// TIA Portal V16 export
// export: Created 2021-11-12T13:31:13.1674631Z, ExportSetting WithDefaults, DisplayName Totally Integrated Automation Portal, DisplayVersion V16 Update 3, DisplayName TIA Portal Version Control Interface, DisplayVersion V16 Update 2, DisplayName TIA Portal Openness, DisplayVersion V16 Update 3, DisplayName SINAMICS Startdrive Advanced, DisplayVersion V16 Update 5, DisplayName SINAMICS Startdrive G130, G150, S120, S150, SINAMICS MV, S210, DisplayVersion V16 Update 5, DisplayName SINAMICS Startdrive G110M, G120, G120C, G120D, G120P, G115D, DisplayVersion V16 Update 5, DisplayName STEP 7 Professional, DisplayVersion V16 Update 3, DisplayName STEP 7 Safety, DisplayVersion V16, DisplayName WinCC UA Professional, DisplayVersion V16 Update 3
FUNCTION_BLOCK "STD_RobotGripper"   // FB1227, LAD
{ S7_Optimized_Access := 'TRUE' }
VERSION : 0.1
// MICE STD Function block
// STD_RobotGripper
// 
// Version      Creation date        Created by
// 1.0                 24.9.2018                   RS
// stored: AutoNumber false, IsIECCheckEnabled false, IsRetainMemResEnabled false, MemoryReserve 100, SetENOAutomatically false, UDAEnableTagReadback false
   VAR_INPUT
      IS_Gripper : "UDT_RobotGripper_Inputs";
      IS_ZoneM { ExternalAccessible := 'False'; ExternalVisible := 'False'; ExternalWritable := 'False'} : "UDT_Status_main";   // Main structure from zone
      IS_ZoneS { ExternalAccessible := 'False'; ExternalVisible := 'False'; ExternalWritable := 'False'} : "UDT_Zone_Status_specific";   // Specific structure from zone
      IB1AlarmSuppress : Bool;   // Suppress alarms
      IT_AckPulseTime : Time := T#200ms;   // Acknowledge pulse length
   END_VAR
   VAR_OUTPUT
      OS_Status : Struct
         Main : "UDT_Status_main";
         Specific : "UDT_RobotGripper_Status_specific";
         Error : "UDT_Error10";
      END_STRUCT;
      OS_Gripper : "UDT_RobotGripper_Outputs";
   END_VAR
   VAR_IN_OUT
      XS_Command : "UDT_RobotGripper_Command";
      XS_Parameter : "UDT_RobotGripper_Parameter";
   END_VAR
   VAR
      SS_Alarm : Struct   // Device alarms / Alarmy zařízení
         MediaNotOK : Bool;   // Gripper media is not OK / Chyba gripperu - nesoulad mezi skutečným a očekávaným stavem
         Res_00_1 : Bool;   // Chyba kontroléru robota - více informací lze nalézt na teachpendantu robota
         Res_00_2 : Bool;   // Chyba robota - více informací lze nalézt na teachpendantu robota
         Res_00_3 : Bool;   // Stisknuto tlačítko Estop na robotu
         Res_00_4 : Bool;   // Bezpečnostní okruh robota přerušen
         Res_00_5 : Bool;   // Motion supervision detekovat kolizi robota
         Res_00_6 : Bool;   // Zpětná vazba čísla úlohy robota neodpovídá požadavku
         Res_00_7 : Bool;   // Zpětná vazba čísla typu úlohy robota neodpovídá požadavku
         Res_01_0 : Bool;
         Res_01_1 : Bool;
         Res_01_2 : Bool;
         Res_01_3 : Bool;
         Res_01_4 : Bool;
         Res_01_5 : Bool;
         Res_01_6 : Bool;
         Res_01_7 : Bool;
      END_STRUCT;
      SS_Warning : Struct   // Device warnings / Varovaní zařízení
         GripperError : Bool;   // Gripper - discrepancy between real and expected state / Chyba gripperu - nesoulad mezi skutečným a očekávaným stavem
         IgnoreGripperError : Bool;   // Gripper error not evaluated / Rychlost robota je omezena na bezpečnou (250mm/s)
         Res_00_2 : Bool;   // Varování robota - více informací lze nalézt na teachpendantu robota
         Res_00_3 : Bool;   // Dialogové okno na Teachpendantu vyžaduje interakci uživatele
         Res_00_4 : Bool;
         Res_00_5 : Bool;
         Res_00_6 : Bool;
         Res_00_7 : Bool;
         Res_01_0 : Bool;
         Res_01_1 : Bool;
         Res_01_2 : Bool;
         Res_01_3 : Bool;
         Res_01_4 : Bool;
         Res_01_5 : Bool;
         Res_01_6 : Bool;
         Res_01_7 : Bool;
         Positive_00_00 : Bool;   // Gripper signal 0 missing
         Positive_00_01 : Bool;   // Gripper signal 1 missing
         Positive_00_02 : Bool;   // Gripper signal 2 missing
         Positive_00_03 : Bool;   // Gripper signal 3 missing
         Positive_00_04 : Bool;   // Gripper signal 4 missing
         Positive_00_05 : Bool;   // Gripper signal 5 missing
         Positive_00_06 : Bool;   // Gripper signal 6 missing
         Positive_00_07 : Bool;   // Gripper signal 7 missing
         Positive_00_08 : Bool;   // Gripper signal 8 missing
         Positive_00_09 : Bool;   // Gripper signal 9 missing
         Positive_00_10 : Bool;   // Gripper signal 10 missing
         Positive_00_11 : Bool;   // Gripper signal 11 missing
         Positive_00_12 : Bool;   // Gripper signal 12 missing
         Positive_00_13 : Bool;   // Gripper signal 13 missing
         Positive_00_14 : Bool;   // Gripper signal 14 missing
         Positive_00_15 : Bool;   // Gripper signal 15 missing
         Positive_00_16 : Bool;   // Gripper signal 16 missing
         Positive_00_17 : Bool;   // Gripper signal 17 missing
         Positive_00_18 : Bool;   // Gripper signal 18 missing
         Positive_00_19 : Bool;   // Gripper signal 19 missing
         Positive_00_20 : Bool;   // Gripper signal 20 missing
         Positive_00_21 : Bool;   // Gripper signal 21 missing
         Positive_00_22 : Bool;   // Gripper signal 22 missing
         Positive_00_23 : Bool;   // Gripper signal 23 missing
         Positive_00_24 : Bool;   // Gripper signal 24 missing
         Positive_00_25 : Bool;   // Gripper signal 25 missing
         Positive_00_26 : Bool;   // Gripper signal 26 missing
         Positive_00_27 : Bool;   // Gripper signal 27 missing
         Positive_00_28 : Bool;   // Gripper signal 28 missing
         Positive_00_29 : Bool;   // Gripper signal 29 missing
         Positive_00_30 : Bool;   // Gripper signal 30 missing
         Positive_00_31 : Bool;   // Gripper signal 31 missing
         Negative_00_00 : Bool;   // Gripper signal 0 is true
         Negative_00_01 : Bool;   // Gripper signal 1 is true
         Negative_00_02 : Bool;   // Gripper signal 2 is true
         Negative_00_03 : Bool;   // Gripper signal 3 is true
         Negative_00_04 : Bool;   // Gripper signal 4 is true
         Negative_00_05 : Bool;   // Gripper signal 5 is true
         Negative_00_06 : Bool;   // Gripper signal 6 is true
         Negative_00_07 : Bool;   // Gripper signal 7 is true
         Negative_00_08 : Bool;   // Gripper signal 8 is true
         Negative_00_09 : Bool;   // Gripper signal 9 is true
         Negative_00_10 : Bool;   // Gripper signal 10 is true
         Negative_00_11 : Bool;   // Gripper signal 11 is true
         Negative_00_12 : Bool;   // Gripper signal 12 is true
         Negative_00_13 : Bool;   // Gripper signal 13 is true
         Negative_00_14 : Bool;   // Gripper signal 14 is true
         Negative_00_15 : Bool;   // Gripper signal 15 is true
         Negative_00_16 : Bool;   // Gripper signal 16 is true
         Negative_00_17 : Bool;   // Gripper signal 17 is true
         Negative_00_18 : Bool;   // Gripper signal 18 is true
         Negative_00_19 : Bool;   // Gripper signal 19 is true
         Negative_00_20 : Bool;   // Gripper signal 20 is true
         Negative_00_21 : Bool;   // Gripper signal 21 is true
         Negative_00_22 : Bool;   // Gripper signal 22 is true
         Negative_00_23 : Bool;   // Gripper signal 23 is true
         Negative_00_24 : Bool;   // Gripper signal 24 is true
         Negative_00_25 : Bool;   // Gripper signal 25 is true
         Negative_00_26 : Bool;   // Gripper signal 26 is true
         Negative_00_27 : Bool;   // Gripper signal 27 is true
         Negative_00_28 : Bool;   // Gripper signal 28 is true
         Negative_00_29 : Bool;   // Gripper signal 29 is true
         Negative_00_30 : Bool;   // Gripper signal 30 is true
         Negative_00_31 : Bool;   // Gripper signal 31 is true
      END_STRUCT;
      SS_Input : Struct
         Gripper { S7_SetPoint := 'True'} : "UDT_RobotGripper_Inputs";
      END_STRUCT;
      SS_Output : Struct
         Gripper { S7_SetPoint := 'True'} : "UDT_RobotGripper_Outputs";
      END_STRUCT;
      SB1IgnoreGripperError : Bool;
      ST_ResetError_TOF { S7_SetPoint := 'True'} : TOF_TIME;
      ST_ResetError_TP { S7_SetPoint := 'True'} : TP_TIME;
      ST_Retest_TOF { S7_SetPoint := 'True'} : TOF_TIME;
      ST_Retry_TOF { S7_SetPoint := 'True'} : TOF_TIME;
   END_VAR
   VAR_TEMP
      TS_Status : Struct
         Main : "UDT_Status_main";
         Specific : "UDT_RobotGripper_Status_specific";
         Error : "UDT_Error10";
      END_STRUCT;
      TS_Parameter : "UDT_RobotGripper_Parameter";
      TS_Command : "UDT_RobotGripper_Command";
      TB1AckPulse : Bool;
      TD_XOR : DWord;
   END_VAR
   VAR_TEMP   // added for the SCL form of the ladder/FBD networks
      _w1 : Bool;
      _w2 : Bool;
      _w3 : Bool;
      _w4 : Bool;
      _w5 : Bool;
      _w6 : Bool;
      _w7 : Bool;
      _w8 : Bool;
      _w9 : Bool;
      _w10 : Bool;
      _w11 : Bool;
      _w12 : Bool;
      _w13 : Bool;
      _w14 : Bool;
      _w15 : Bool;
      _w16 : Bool;
      _w17 : Bool;
      _w18 : Bool;
      _w19 : Bool;
      _w20 : Bool;
      _w21 : Bool;
      _w22 : Bool;
      _w23 : Bool;
      _w24 : Bool;
      _w25 : Bool;
      _w26 : Bool;
      _w27 : Bool;
      _w28 : Bool;
      _w29 : Bool;
      _w30 : Bool;
      _w31 : Bool;
      _w32 : Bool;
   END_VAR
BEGIN

REGION Network 1: Clear temporary TS_Status - Main, Specific
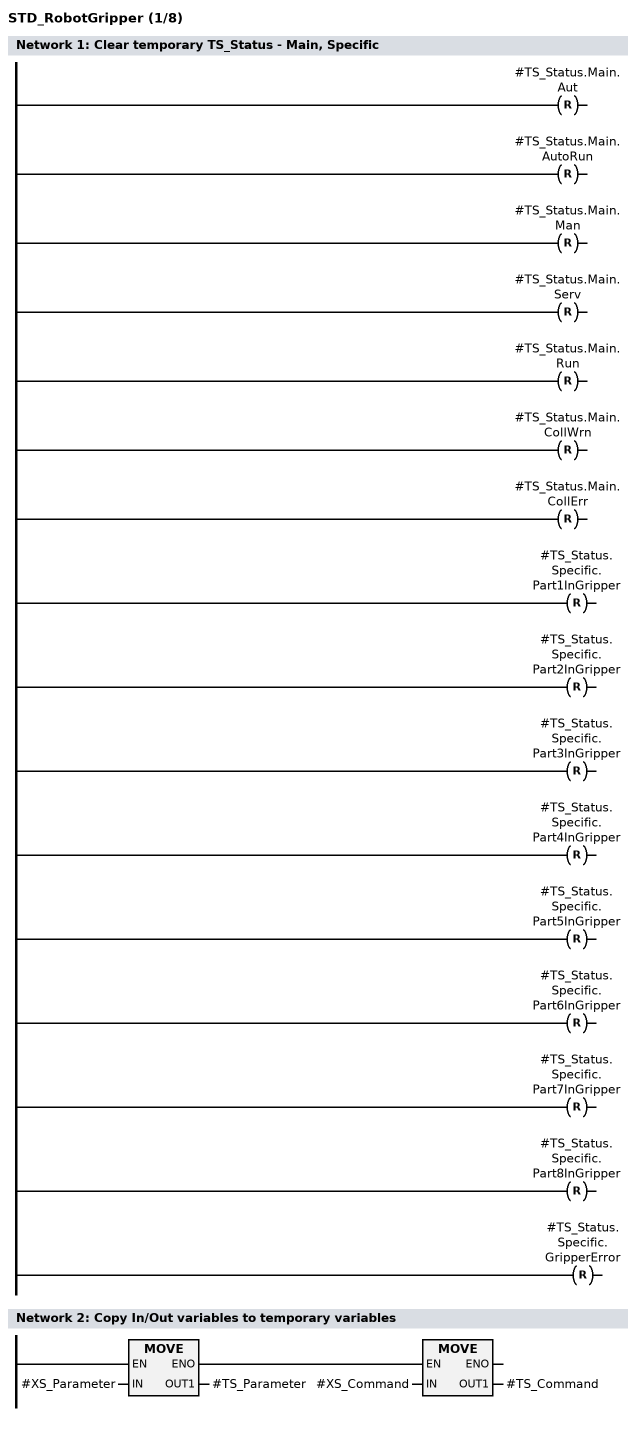
   RUNG wire#powerrail
      R_Coil( #TS_Status.Main.Aut )
   END_RUNG
   RUNG wire#powerrail
      R_Coil( #TS_Status.Main.AutoRun )
   END_RUNG
   RUNG wire#powerrail
      R_Coil( #TS_Status.Main.Man )
   END_RUNG
   RUNG wire#powerrail
      R_Coil( #TS_Status.Main.Serv )
   END_RUNG
   RUNG wire#powerrail
      R_Coil( #TS_Status.Main.Run )
   END_RUNG
   RUNG wire#powerrail
      R_Coil( #TS_Status.Main.CollWrn )
   END_RUNG
   RUNG wire#powerrail
      R_Coil( #TS_Status.Main.CollErr )
   END_RUNG
   RUNG wire#powerrail
      R_Coil( #TS_Status.Specific.Part1InGripper )
   END_RUNG
   RUNG wire#powerrail
      R_Coil( #TS_Status.Specific.Part2InGripper )
   END_RUNG
   RUNG wire#powerrail
      R_Coil( #TS_Status.Specific.Part3InGripper )
   END_RUNG
   RUNG wire#powerrail
      R_Coil( #TS_Status.Specific.Part4InGripper )
   END_RUNG
   RUNG wire#powerrail
      R_Coil( #TS_Status.Specific.Part5InGripper )
   END_RUNG
   RUNG wire#powerrail
      R_Coil( #TS_Status.Specific.Part6InGripper )
   END_RUNG
   RUNG wire#powerrail
      R_Coil( #TS_Status.Specific.Part7InGripper )
   END_RUNG
   RUNG wire#powerrail
      R_Coil( #TS_Status.Specific.Part8InGripper )
   END_RUNG
   RUNG wire#powerrail
      R_Coil( #TS_Status.Specific.GripperError )
   END_RUNG
   // the same network as SCL:
   #TS_Status.Main.Aut := FALSE;
   #TS_Status.Main.AutoRun := FALSE;
   #TS_Status.Main.Man := FALSE;
   #TS_Status.Main.Serv := FALSE;
   #TS_Status.Main.Run := FALSE;
   #TS_Status.Main.CollWrn := FALSE;
   #TS_Status.Main.CollErr := FALSE;
   #TS_Status.Specific.Part1InGripper := FALSE;
   #TS_Status.Specific.Part2InGripper := FALSE;
   #TS_Status.Specific.Part3InGripper := FALSE;
   #TS_Status.Specific.Part4InGripper := FALSE;
   #TS_Status.Specific.Part5InGripper := FALSE;
   #TS_Status.Specific.Part6InGripper := FALSE;
   #TS_Status.Specific.Part7InGripper := FALSE;
   #TS_Status.Specific.Part8InGripper := FALSE;
   #TS_Status.Specific.GripperError := FALSE;
END_REGION

REGION Network 2: Copy In/Out variables to temporary variables
   RUNG wire#powerrail
      Move(in := #XS_Parameter, out1 => #TS_Parameter)
      Move(in := #XS_Command, out1 => #TS_Command)
   END_RUNG
   // the same network as SCL:
   #TS_Parameter := #XS_Parameter;
   #TS_Command := #XS_Command;
END_REGION

REGION Network 3: Read data from Robot Interface
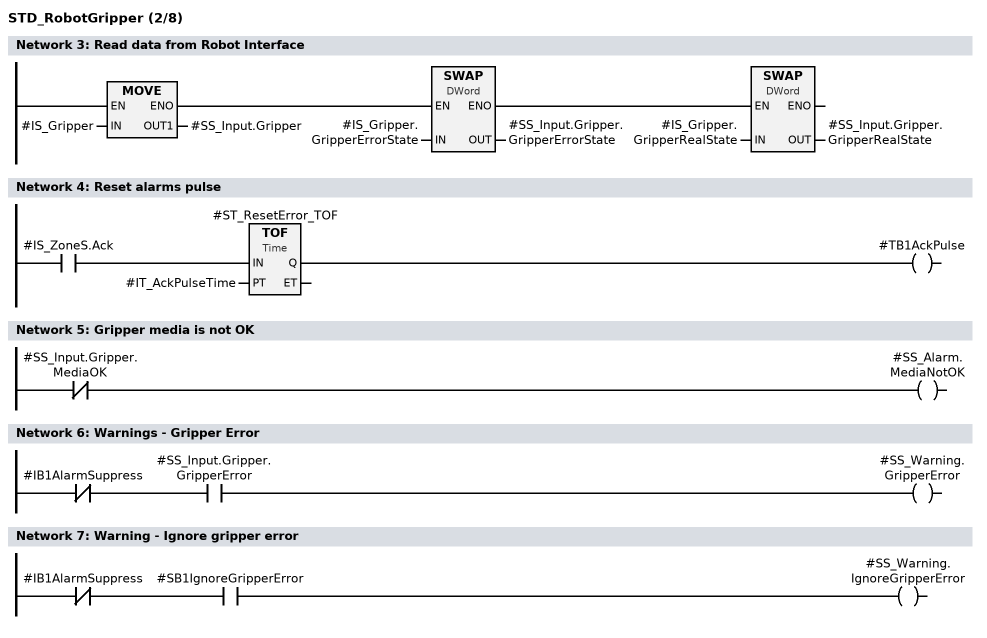
   #SS_Input.Gripper := #IS_Gripper;
   #SS_Input.Gripper.GripperErrorState := SWAP(#IS_Gripper.GripperErrorState);
   #SS_Input.Gripper.GripperRealState := SWAP(#IS_Gripper.GripperRealState);
END_REGION

REGION Network 4: Reset alarms pulse
   RUNG wire#powerrail
      Contact( #IS_ZoneS.Ack )
      { S7_Templates := "time_type := Time" } #ST_ResetError_TOF.TOF(pt := #IT_AckPulseTime, et =>)
      Coil( #TB1AckPulse )
   END_RUNG
   // the same network as SCL:
   #ST_ResetError_TOF(IN := #IS_ZoneS.Ack, PT := #IT_AckPulseTime);   // TOF
   #TB1AckPulse := #ST_ResetError_TOF.Q;
END_REGION

REGION Network 5: Gripper media is not OK
   RUNG wire#powerrail
      I_Contact( #SS_Input.Gripper.MediaOK )
      Coil( #SS_Alarm.MediaNotOK )
   END_RUNG
   // the same network as SCL:
   #SS_Alarm.MediaNotOK := NOT #SS_Input.Gripper.MediaOK;
END_REGION

REGION Network 6: Warnings - Gripper Error
   RUNG wire#powerrail
      I_Contact( #IB1AlarmSuppress )
      Contact( #SS_Input.Gripper.GripperError )
      Coil( #SS_Warning.GripperError )
   END_RUNG
   // the same network as SCL:
   #SS_Warning.GripperError := NOT #IB1AlarmSuppress AND #SS_Input.Gripper.GripperError;
END_REGION

REGION Network 7: Warning - Ignore gripper error
   RUNG wire#powerrail
      I_Contact( #IB1AlarmSuppress )
      Contact( #SB1IgnoreGripperError )
      Coil( #SS_Warning.IgnoreGripperError )
   END_RUNG
   // the same network as SCL:
   #SS_Warning.IgnoreGripperError := NOT #IB1AlarmSuppress AND #SB1IgnoreGripperError;
END_REGION

REGION Network 8: Gripper Specific error
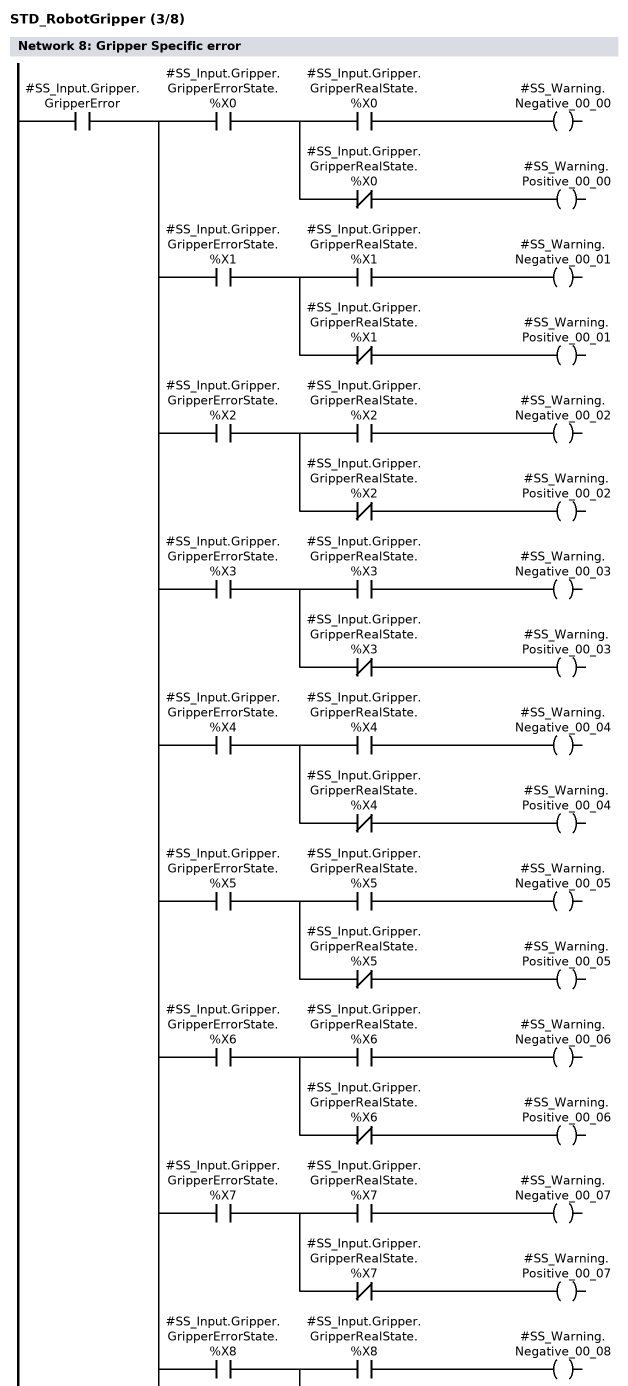
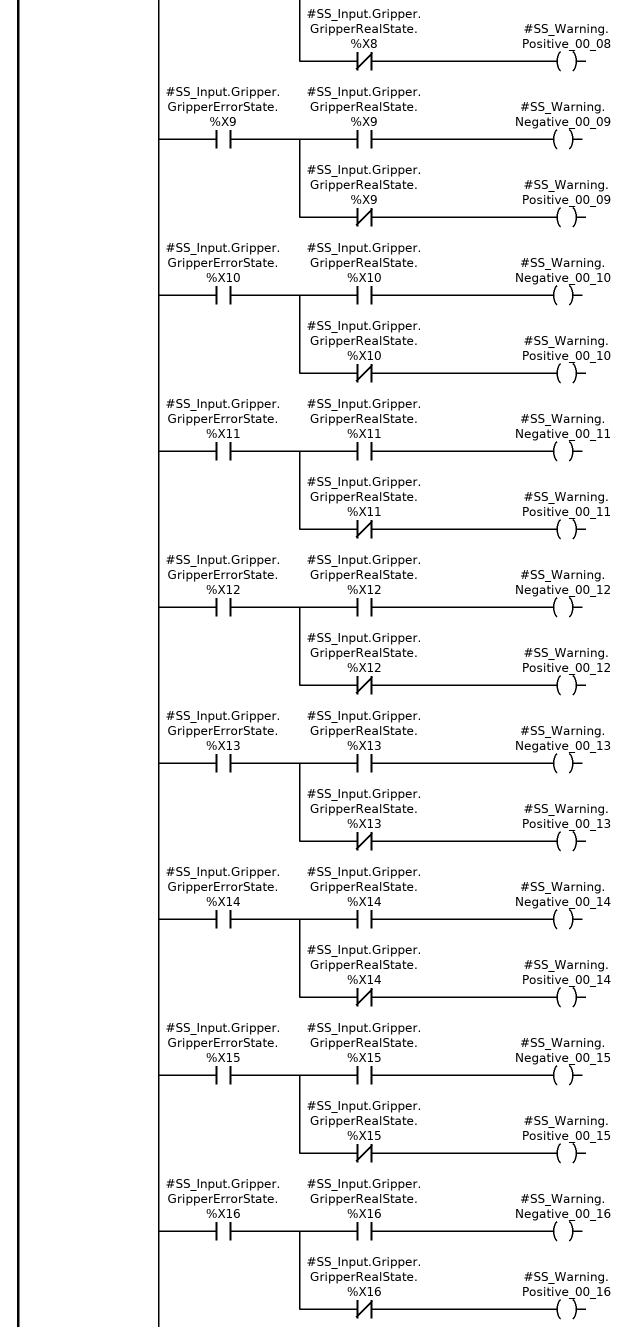
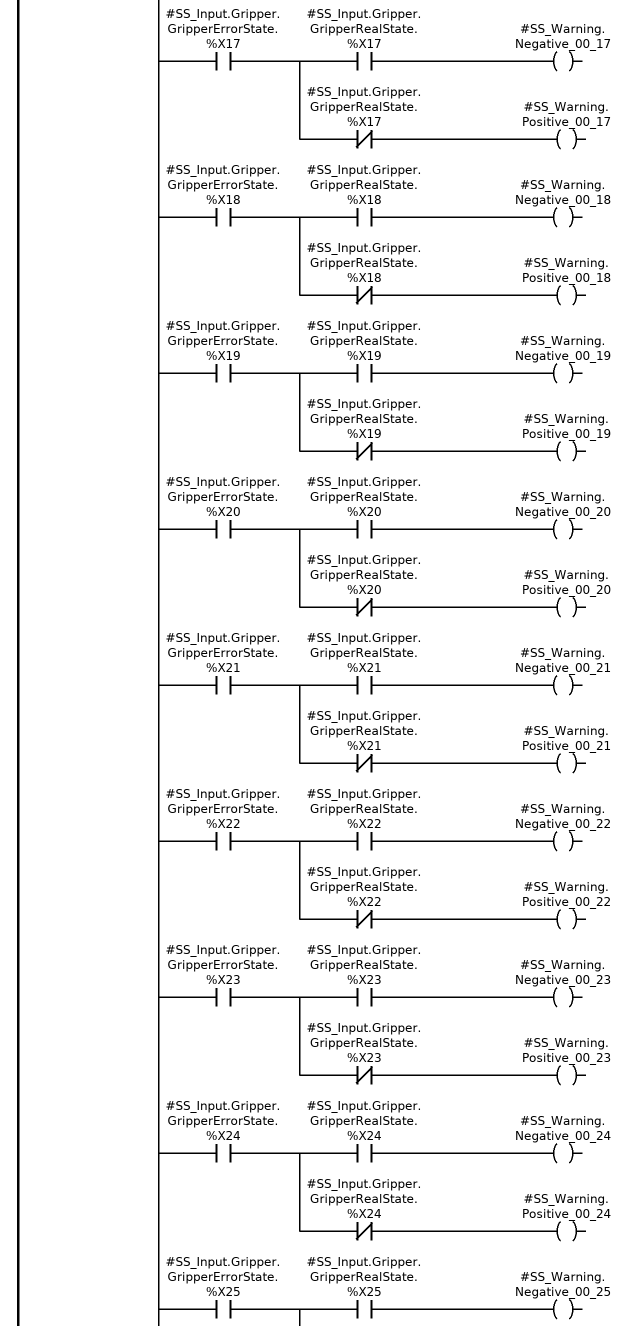
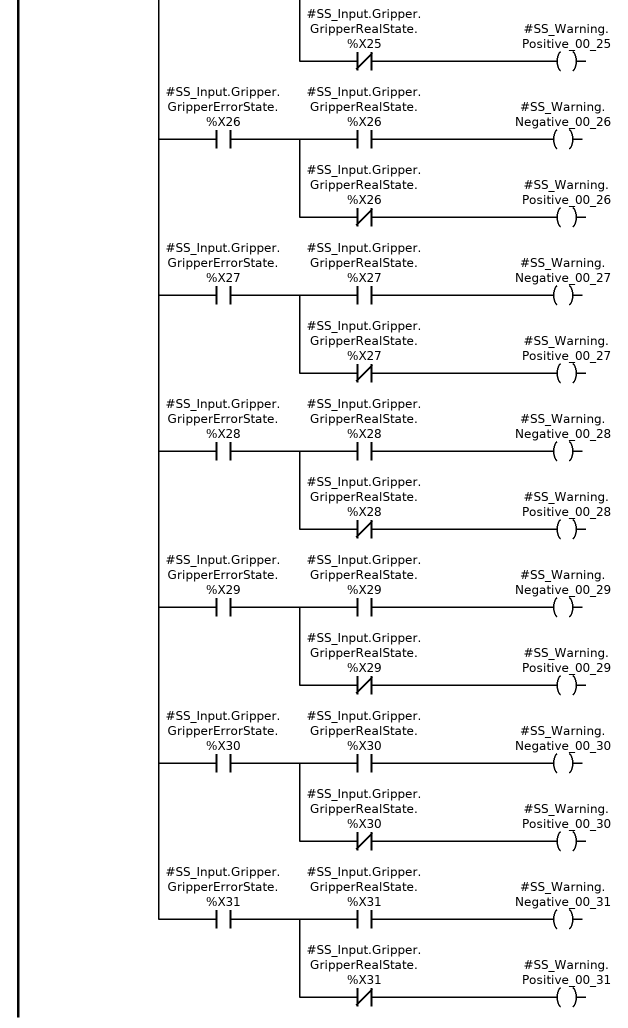
   RUNG wire#powerrail
      Contact( #SS_Input.Gripper.GripperError )
      wire#w1
      Contact( #SS_Input.Gripper.GripperErrorState.%X0 )
      wire#w2
      Contact( #SS_Input.Gripper.GripperRealState.%X0 )
      Coil( #SS_Warning.Negative_00_00 )
   END_RUNG
   RUNG wire#w2
      I_Contact( #SS_Input.Gripper.GripperRealState.%X0 )
      Coil( #SS_Warning.Positive_00_00 )
   END_RUNG
   RUNG wire#w1
      Contact( #SS_Input.Gripper.GripperErrorState.%X1 )
      wire#w3
      Contact( #SS_Input.Gripper.GripperRealState.%X1 )
      Coil( #SS_Warning.Negative_00_01 )
   END_RUNG
   RUNG wire#w3
      I_Contact( #SS_Input.Gripper.GripperRealState.%X1 )
      Coil( #SS_Warning.Positive_00_01 )
   END_RUNG
   RUNG wire#w1
      Contact( #SS_Input.Gripper.GripperErrorState.%X2 )
      wire#w4
      Contact( #SS_Input.Gripper.GripperRealState.%X2 )
      Coil( #SS_Warning.Negative_00_02 )
   END_RUNG
   RUNG wire#w4
      I_Contact( #SS_Input.Gripper.GripperRealState.%X2 )
      Coil( #SS_Warning.Positive_00_02 )
   END_RUNG
   RUNG wire#w1
      Contact( #SS_Input.Gripper.GripperErrorState.%X3 )
      wire#w5
      Contact( #SS_Input.Gripper.GripperRealState.%X3 )
      Coil( #SS_Warning.Negative_00_03 )
   END_RUNG
   RUNG wire#w5
      I_Contact( #SS_Input.Gripper.GripperRealState.%X3 )
      Coil( #SS_Warning.Positive_00_03 )
   END_RUNG
   RUNG wire#w1
      Contact( #SS_Input.Gripper.GripperErrorState.%X4 )
      wire#w6
      Contact( #SS_Input.Gripper.GripperRealState.%X4 )
      Coil( #SS_Warning.Negative_00_04 )
   END_RUNG
   RUNG wire#w6
      I_Contact( #SS_Input.Gripper.GripperRealState.%X4 )
      Coil( #SS_Warning.Positive_00_04 )
   END_RUNG
   RUNG wire#w1
      Contact( #SS_Input.Gripper.GripperErrorState.%X5 )
      wire#w7
      Contact( #SS_Input.Gripper.GripperRealState.%X5 )
      Coil( #SS_Warning.Negative_00_05 )
   END_RUNG
   RUNG wire#w7
      I_Contact( #SS_Input.Gripper.GripperRealState.%X5 )
      Coil( #SS_Warning.Positive_00_05 )
   END_RUNG
   RUNG wire#w1
      Contact( #SS_Input.Gripper.GripperErrorState.%X6 )
      wire#w8
      Contact( #SS_Input.Gripper.GripperRealState.%X6 )
      Coil( #SS_Warning.Negative_00_06 )
   END_RUNG
   RUNG wire#w8
      I_Contact( #SS_Input.Gripper.GripperRealState.%X6 )
      Coil( #SS_Warning.Positive_00_06 )
   END_RUNG
   RUNG wire#w1
      Contact( #SS_Input.Gripper.GripperErrorState.%X7 )
      wire#w9
      Contact( #SS_Input.Gripper.GripperRealState.%X7 )
      Coil( #SS_Warning.Negative_00_07 )
   END_RUNG
   RUNG wire#w9
      I_Contact( #SS_Input.Gripper.GripperRealState.%X7 )
      Coil( #SS_Warning.Positive_00_07 )
   END_RUNG
   RUNG wire#w1
      Contact( #SS_Input.Gripper.GripperErrorState.%X8 )
      wire#w10
      Contact( #SS_Input.Gripper.GripperRealState.%X8 )
      Coil( #SS_Warning.Negative_00_08 )
   END_RUNG
   RUNG wire#w10
      I_Contact( #SS_Input.Gripper.GripperRealState.%X8 )
      Coil( #SS_Warning.Positive_00_08 )
   END_RUNG
   RUNG wire#w1
      Contact( #SS_Input.Gripper.GripperErrorState.%X9 )
      wire#w11
      Contact( #SS_Input.Gripper.GripperRealState.%X9 )
      Coil( #SS_Warning.Negative_00_09 )
   END_RUNG
   RUNG wire#w11
      I_Contact( #SS_Input.Gripper.GripperRealState.%X9 )
      Coil( #SS_Warning.Positive_00_09 )
   END_RUNG
   RUNG wire#w1
      Contact( #SS_Input.Gripper.GripperErrorState.%X10 )
      wire#w12
      Contact( #SS_Input.Gripper.GripperRealState.%X10 )
      Coil( #SS_Warning.Negative_00_10 )
   END_RUNG
   RUNG wire#w12
      I_Contact( #SS_Input.Gripper.GripperRealState.%X10 )
      Coil( #SS_Warning.Positive_00_10 )
   END_RUNG
   RUNG wire#w1
      Contact( #SS_Input.Gripper.GripperErrorState.%X11 )
      wire#w13
      Contact( #SS_Input.Gripper.GripperRealState.%X11 )
      Coil( #SS_Warning.Negative_00_11 )
   END_RUNG
   RUNG wire#w13
      I_Contact( #SS_Input.Gripper.GripperRealState.%X11 )
      Coil( #SS_Warning.Positive_00_11 )
   END_RUNG
   RUNG wire#w1
      Contact( #SS_Input.Gripper.GripperErrorState.%X12 )
      wire#w14
      Contact( #SS_Input.Gripper.GripperRealState.%X12 )
      Coil( #SS_Warning.Negative_00_12 )
   END_RUNG
   RUNG wire#w14
      I_Contact( #SS_Input.Gripper.GripperRealState.%X12 )
      Coil( #SS_Warning.Positive_00_12 )
   END_RUNG
   RUNG wire#w1
      Contact( #SS_Input.Gripper.GripperErrorState.%X13 )
      wire#w15
      Contact( #SS_Input.Gripper.GripperRealState.%X13 )
      Coil( #SS_Warning.Negative_00_13 )
   END_RUNG
   RUNG wire#w15
      I_Contact( #SS_Input.Gripper.GripperRealState.%X13 )
      Coil( #SS_Warning.Positive_00_13 )
   END_RUNG
   RUNG wire#w1
      Contact( #SS_Input.Gripper.GripperErrorState.%X14 )
      wire#w16
      Contact( #SS_Input.Gripper.GripperRealState.%X14 )
      Coil( #SS_Warning.Negative_00_14 )
   END_RUNG
   RUNG wire#w16
      I_Contact( #SS_Input.Gripper.GripperRealState.%X14 )
      Coil( #SS_Warning.Positive_00_14 )
   END_RUNG
   RUNG wire#w1
      Contact( #SS_Input.Gripper.GripperErrorState.%X15 )
      wire#w17
      Contact( #SS_Input.Gripper.GripperRealState.%X15 )
      Coil( #SS_Warning.Negative_00_15 )
   END_RUNG
   RUNG wire#w17
      I_Contact( #SS_Input.Gripper.GripperRealState.%X15 )
      Coil( #SS_Warning.Positive_00_15 )
   END_RUNG
   RUNG wire#w1
      Contact( #SS_Input.Gripper.GripperErrorState.%X16 )
      wire#w18
      Contact( #SS_Input.Gripper.GripperRealState.%X16 )
      Coil( #SS_Warning.Negative_00_16 )
   END_RUNG
   RUNG wire#w18
      I_Contact( #SS_Input.Gripper.GripperRealState.%X16 )
      Coil( #SS_Warning.Positive_00_16 )
   END_RUNG
   RUNG wire#w1
      Contact( #SS_Input.Gripper.GripperErrorState.%X17 )
      wire#w19
      Contact( #SS_Input.Gripper.GripperRealState.%X17 )
      Coil( #SS_Warning.Negative_00_17 )
   END_RUNG
   RUNG wire#w19
      I_Contact( #SS_Input.Gripper.GripperRealState.%X17 )
      Coil( #SS_Warning.Positive_00_17 )
   END_RUNG
   RUNG wire#w1
      Contact( #SS_Input.Gripper.GripperErrorState.%X18 )
      wire#w20
      Contact( #SS_Input.Gripper.GripperRealState.%X18 )
      Coil( #SS_Warning.Negative_00_18 )
   END_RUNG
   RUNG wire#w20
      I_Contact( #SS_Input.Gripper.GripperRealState.%X18 )
      Coil( #SS_Warning.Positive_00_18 )
   END_RUNG
   RUNG wire#w1
      Contact( #SS_Input.Gripper.GripperErrorState.%X19 )
      wire#w21
      Contact( #SS_Input.Gripper.GripperRealState.%X19 )
      Coil( #SS_Warning.Negative_00_19 )
   END_RUNG
   RUNG wire#w21
      I_Contact( #SS_Input.Gripper.GripperRealState.%X19 )
      Coil( #SS_Warning.Positive_00_19 )
   END_RUNG
   RUNG wire#w1
      Contact( #SS_Input.Gripper.GripperErrorState.%X20 )
      wire#w22
      Contact( #SS_Input.Gripper.GripperRealState.%X20 )
      Coil( #SS_Warning.Negative_00_20 )
   END_RUNG
   RUNG wire#w22
      I_Contact( #SS_Input.Gripper.GripperRealState.%X20 )
      Coil( #SS_Warning.Positive_00_20 )
   END_RUNG
   RUNG wire#w1
      Contact( #SS_Input.Gripper.GripperErrorState.%X21 )
      wire#w23
      Contact( #SS_Input.Gripper.GripperRealState.%X21 )
      Coil( #SS_Warning.Negative_00_21 )
   END_RUNG
   RUNG wire#w23
      I_Contact( #SS_Input.Gripper.GripperRealState.%X21 )
      Coil( #SS_Warning.Positive_00_21 )
   END_RUNG
   RUNG wire#w1
      Contact( #SS_Input.Gripper.GripperErrorState.%X22 )
      wire#w24
      Contact( #SS_Input.Gripper.GripperRealState.%X22 )
      Coil( #SS_Warning.Negative_00_22 )
   END_RUNG
   RUNG wire#w24
      I_Contact( #SS_Input.Gripper.GripperRealState.%X22 )
      Coil( #SS_Warning.Positive_00_22 )
   END_RUNG
   RUNG wire#w1
      Contact( #SS_Input.Gripper.GripperErrorState.%X23 )
      wire#w25
      Contact( #SS_Input.Gripper.GripperRealState.%X23 )
      Coil( #SS_Warning.Negative_00_23 )
   END_RUNG
   RUNG wire#w25
      I_Contact( #SS_Input.Gripper.GripperRealState.%X23 )
      Coil( #SS_Warning.Positive_00_23 )
   END_RUNG
   RUNG wire#w1
      Contact( #SS_Input.Gripper.GripperErrorState.%X24 )
      wire#w26
      Contact( #SS_Input.Gripper.GripperRealState.%X24 )
      Coil( #SS_Warning.Negative_00_24 )
   END_RUNG
   RUNG wire#w26
      I_Contact( #SS_Input.Gripper.GripperRealState.%X24 )
      Coil( #SS_Warning.Positive_00_24 )
   END_RUNG
   RUNG wire#w1
      Contact( #SS_Input.Gripper.GripperErrorState.%X25 )
      wire#w27
      Contact( #SS_Input.Gripper.GripperRealState.%X25 )
      Coil( #SS_Warning.Negative_00_25 )
   END_RUNG
   RUNG wire#w27
      I_Contact( #SS_Input.Gripper.GripperRealState.%X25 )
      Coil( #SS_Warning.Positive_00_25 )
   END_RUNG
   RUNG wire#w1
      Contact( #SS_Input.Gripper.GripperErrorState.%X26 )
      wire#w28
      Contact( #SS_Input.Gripper.GripperRealState.%X26 )
      Coil( #SS_Warning.Negative_00_26 )
   END_RUNG
   RUNG wire#w28
      I_Contact( #SS_Input.Gripper.GripperRealState.%X26 )
      Coil( #SS_Warning.Positive_00_26 )
   END_RUNG
   RUNG wire#w1
      Contact( #SS_Input.Gripper.GripperErrorState.%X27 )
      wire#w29
      Contact( #SS_Input.Gripper.GripperRealState.%X27 )
      Coil( #SS_Warning.Negative_00_27 )
   END_RUNG
   RUNG wire#w29
      I_Contact( #SS_Input.Gripper.GripperRealState.%X27 )
      Coil( #SS_Warning.Positive_00_27 )
   END_RUNG
   RUNG wire#w1
      Contact( #SS_Input.Gripper.GripperErrorState.%X28 )
      wire#w30
      Contact( #SS_Input.Gripper.GripperRealState.%X28 )
      Coil( #SS_Warning.Negative_00_28 )
   END_RUNG
   RUNG wire#w30
      I_Contact( #SS_Input.Gripper.GripperRealState.%X28 )
      Coil( #SS_Warning.Positive_00_28 )
   END_RUNG
   RUNG wire#w1
      Contact( #SS_Input.Gripper.GripperErrorState.%X29 )
      wire#w31
      Contact( #SS_Input.Gripper.GripperRealState.%X29 )
      Coil( #SS_Warning.Negative_00_29 )
   END_RUNG
   RUNG wire#w31
      I_Contact( #SS_Input.Gripper.GripperRealState.%X29 )
      Coil( #SS_Warning.Positive_00_29 )
   END_RUNG
   RUNG wire#w1
      Contact( #SS_Input.Gripper.GripperErrorState.%X30 )
      wire#w32
      Contact( #SS_Input.Gripper.GripperRealState.%X30 )
      Coil( #SS_Warning.Negative_00_30 )
   END_RUNG
   RUNG wire#w32
      I_Contact( #SS_Input.Gripper.GripperRealState.%X30 )
      Coil( #SS_Warning.Positive_00_30 )
   END_RUNG
   RUNG wire#w1
      Contact( #SS_Input.Gripper.GripperErrorState.%X31 )
      wire#w33
      Contact( #SS_Input.Gripper.GripperRealState.%X31 )
      Coil( #SS_Warning.Negative_00_31 )
   END_RUNG
   RUNG wire#w33
      I_Contact( #SS_Input.Gripper.GripperRealState.%X31 )
      Coil( #SS_Warning.Positive_00_31 )
   END_RUNG
   // the same network as SCL:
   #_w1 := #SS_Input.Gripper.GripperError AND #SS_Input.Gripper.GripperErrorState.%X0;
   #SS_Warning.Negative_00_00 := #_w1 AND #SS_Input.Gripper.GripperRealState.%X0;
   #SS_Warning.Positive_00_00 := #_w1 AND NOT #SS_Input.Gripper.GripperRealState.%X0;
   #_w2 := #SS_Input.Gripper.GripperError AND #SS_Input.Gripper.GripperErrorState.%X1;
   #SS_Warning.Negative_00_01 := #_w2 AND #SS_Input.Gripper.GripperRealState.%X1;
   #SS_Warning.Positive_00_01 := #_w2 AND NOT #SS_Input.Gripper.GripperRealState.%X1;
   #_w3 := #SS_Input.Gripper.GripperError AND #SS_Input.Gripper.GripperErrorState.%X2;
   #SS_Warning.Negative_00_02 := #_w3 AND #SS_Input.Gripper.GripperRealState.%X2;
   #SS_Warning.Positive_00_02 := #_w3 AND NOT #SS_Input.Gripper.GripperRealState.%X2;
   #_w4 := #SS_Input.Gripper.GripperError AND #SS_Input.Gripper.GripperErrorState.%X3;
   #SS_Warning.Negative_00_03 := #_w4 AND #SS_Input.Gripper.GripperRealState.%X3;
   #SS_Warning.Positive_00_03 := #_w4 AND NOT #SS_Input.Gripper.GripperRealState.%X3;
   #_w5 := #SS_Input.Gripper.GripperError AND #SS_Input.Gripper.GripperErrorState.%X4;
   #SS_Warning.Negative_00_04 := #_w5 AND #SS_Input.Gripper.GripperRealState.%X4;
   #SS_Warning.Positive_00_04 := #_w5 AND NOT #SS_Input.Gripper.GripperRealState.%X4;
   #_w6 := #SS_Input.Gripper.GripperError AND #SS_Input.Gripper.GripperErrorState.%X5;
   #SS_Warning.Negative_00_05 := #_w6 AND #SS_Input.Gripper.GripperRealState.%X5;
   #SS_Warning.Positive_00_05 := #_w6 AND NOT #SS_Input.Gripper.GripperRealState.%X5;
   #_w7 := #SS_Input.Gripper.GripperError AND #SS_Input.Gripper.GripperErrorState.%X6;
   #SS_Warning.Negative_00_06 := #_w7 AND #SS_Input.Gripper.GripperRealState.%X6;
   #SS_Warning.Positive_00_06 := #_w7 AND NOT #SS_Input.Gripper.GripperRealState.%X6;
   #_w8 := #SS_Input.Gripper.GripperError AND #SS_Input.Gripper.GripperErrorState.%X7;
   #SS_Warning.Negative_00_07 := #_w8 AND #SS_Input.Gripper.GripperRealState.%X7;
   #SS_Warning.Positive_00_07 := #_w8 AND NOT #SS_Input.Gripper.GripperRealState.%X7;
   #_w9 := #SS_Input.Gripper.GripperError AND #SS_Input.Gripper.GripperErrorState.%X8;
   #SS_Warning.Negative_00_08 := #_w9 AND #SS_Input.Gripper.GripperRealState.%X8;
   #SS_Warning.Positive_00_08 := #_w9 AND NOT #SS_Input.Gripper.GripperRealState.%X8;
   #_w10 := #SS_Input.Gripper.GripperError AND #SS_Input.Gripper.GripperErrorState.%X9;
   #SS_Warning.Negative_00_09 := #_w10 AND #SS_Input.Gripper.GripperRealState.%X9;
   #SS_Warning.Positive_00_09 := #_w10 AND NOT #SS_Input.Gripper.GripperRealState.%X9;
   #_w11 := #SS_Input.Gripper.GripperError AND #SS_Input.Gripper.GripperErrorState.%X10;
   #SS_Warning.Negative_00_10 := #_w11 AND #SS_Input.Gripper.GripperRealState.%X10;
   #SS_Warning.Positive_00_10 := #_w11 AND NOT #SS_Input.Gripper.GripperRealState.%X10;
   #_w12 := #SS_Input.Gripper.GripperError AND #SS_Input.Gripper.GripperErrorState.%X11;
   #SS_Warning.Negative_00_11 := #_w12 AND #SS_Input.Gripper.GripperRealState.%X11;
   #SS_Warning.Positive_00_11 := #_w12 AND NOT #SS_Input.Gripper.GripperRealState.%X11;
   #_w13 := #SS_Input.Gripper.GripperError AND #SS_Input.Gripper.GripperErrorState.%X12;
   #SS_Warning.Negative_00_12 := #_w13 AND #SS_Input.Gripper.GripperRealState.%X12;
   #SS_Warning.Positive_00_12 := #_w13 AND NOT #SS_Input.Gripper.GripperRealState.%X12;
   #_w14 := #SS_Input.Gripper.GripperError AND #SS_Input.Gripper.GripperErrorState.%X13;
   #SS_Warning.Negative_00_13 := #_w14 AND #SS_Input.Gripper.GripperRealState.%X13;
   #SS_Warning.Positive_00_13 := #_w14 AND NOT #SS_Input.Gripper.GripperRealState.%X13;
   #_w15 := #SS_Input.Gripper.GripperError AND #SS_Input.Gripper.GripperErrorState.%X14;
   #SS_Warning.Negative_00_14 := #_w15 AND #SS_Input.Gripper.GripperRealState.%X14;
   #SS_Warning.Positive_00_14 := #_w15 AND NOT #SS_Input.Gripper.GripperRealState.%X14;
   #_w16 := #SS_Input.Gripper.GripperError AND #SS_Input.Gripper.GripperErrorState.%X15;
   #SS_Warning.Negative_00_15 := #_w16 AND #SS_Input.Gripper.GripperRealState.%X15;
   #SS_Warning.Positive_00_15 := #_w16 AND NOT #SS_Input.Gripper.GripperRealState.%X15;
   #_w17 := #SS_Input.Gripper.GripperError AND #SS_Input.Gripper.GripperErrorState.%X16;
   #SS_Warning.Negative_00_16 := #_w17 AND #SS_Input.Gripper.GripperRealState.%X16;
   #SS_Warning.Positive_00_16 := #_w17 AND NOT #SS_Input.Gripper.GripperRealState.%X16;
   #_w18 := #SS_Input.Gripper.GripperError AND #SS_Input.Gripper.GripperErrorState.%X17;
   #SS_Warning.Negative_00_17 := #_w18 AND #SS_Input.Gripper.GripperRealState.%X17;
   #SS_Warning.Positive_00_17 := #_w18 AND NOT #SS_Input.Gripper.GripperRealState.%X17;
   #_w19 := #SS_Input.Gripper.GripperError AND #SS_Input.Gripper.GripperErrorState.%X18;
   #SS_Warning.Negative_00_18 := #_w19 AND #SS_Input.Gripper.GripperRealState.%X18;
   #SS_Warning.Positive_00_18 := #_w19 AND NOT #SS_Input.Gripper.GripperRealState.%X18;
   #_w20 := #SS_Input.Gripper.GripperError AND #SS_Input.Gripper.GripperErrorState.%X19;
   #SS_Warning.Negative_00_19 := #_w20 AND #SS_Input.Gripper.GripperRealState.%X19;
   #SS_Warning.Positive_00_19 := #_w20 AND NOT #SS_Input.Gripper.GripperRealState.%X19;
   #_w21 := #SS_Input.Gripper.GripperError AND #SS_Input.Gripper.GripperErrorState.%X20;
   #SS_Warning.Negative_00_20 := #_w21 AND #SS_Input.Gripper.GripperRealState.%X20;
   #SS_Warning.Positive_00_20 := #_w21 AND NOT #SS_Input.Gripper.GripperRealState.%X20;
   #_w22 := #SS_Input.Gripper.GripperError AND #SS_Input.Gripper.GripperErrorState.%X21;
   #SS_Warning.Negative_00_21 := #_w22 AND #SS_Input.Gripper.GripperRealState.%X21;
   #SS_Warning.Positive_00_21 := #_w22 AND NOT #SS_Input.Gripper.GripperRealState.%X21;
   #_w23 := #SS_Input.Gripper.GripperError AND #SS_Input.Gripper.GripperErrorState.%X22;
   #SS_Warning.Negative_00_22 := #_w23 AND #SS_Input.Gripper.GripperRealState.%X22;
   #SS_Warning.Positive_00_22 := #_w23 AND NOT #SS_Input.Gripper.GripperRealState.%X22;
   #_w24 := #SS_Input.Gripper.GripperError AND #SS_Input.Gripper.GripperErrorState.%X23;
   #SS_Warning.Negative_00_23 := #_w24 AND #SS_Input.Gripper.GripperRealState.%X23;
   #SS_Warning.Positive_00_23 := #_w24 AND NOT #SS_Input.Gripper.GripperRealState.%X23;
   #_w25 := #SS_Input.Gripper.GripperError AND #SS_Input.Gripper.GripperErrorState.%X24;
   #SS_Warning.Negative_00_24 := #_w25 AND #SS_Input.Gripper.GripperRealState.%X24;
   #SS_Warning.Positive_00_24 := #_w25 AND NOT #SS_Input.Gripper.GripperRealState.%X24;
   #_w26 := #SS_Input.Gripper.GripperError AND #SS_Input.Gripper.GripperErrorState.%X25;
   #SS_Warning.Negative_00_25 := #_w26 AND #SS_Input.Gripper.GripperRealState.%X25;
   #SS_Warning.Positive_00_25 := #_w26 AND NOT #SS_Input.Gripper.GripperRealState.%X25;
   #_w27 := #SS_Input.Gripper.GripperError AND #SS_Input.Gripper.GripperErrorState.%X26;
   #SS_Warning.Negative_00_26 := #_w27 AND #SS_Input.Gripper.GripperRealState.%X26;
   #SS_Warning.Positive_00_26 := #_w27 AND NOT #SS_Input.Gripper.GripperRealState.%X26;
   #_w28 := #SS_Input.Gripper.GripperError AND #SS_Input.Gripper.GripperErrorState.%X27;
   #SS_Warning.Negative_00_27 := #_w28 AND #SS_Input.Gripper.GripperRealState.%X27;
   #SS_Warning.Positive_00_27 := #_w28 AND NOT #SS_Input.Gripper.GripperRealState.%X27;
   #_w29 := #SS_Input.Gripper.GripperError AND #SS_Input.Gripper.GripperErrorState.%X28;
   #SS_Warning.Negative_00_28 := #_w29 AND #SS_Input.Gripper.GripperRealState.%X28;
   #SS_Warning.Positive_00_28 := #_w29 AND NOT #SS_Input.Gripper.GripperRealState.%X28;
   #_w30 := #SS_Input.Gripper.GripperError AND #SS_Input.Gripper.GripperErrorState.%X29;
   #SS_Warning.Negative_00_29 := #_w30 AND #SS_Input.Gripper.GripperRealState.%X29;
   #SS_Warning.Positive_00_29 := #_w30 AND NOT #SS_Input.Gripper.GripperRealState.%X29;
   #_w31 := #SS_Input.Gripper.GripperError AND #SS_Input.Gripper.GripperErrorState.%X30;
   #SS_Warning.Negative_00_30 := #_w31 AND #SS_Input.Gripper.GripperRealState.%X30;
   #SS_Warning.Positive_00_30 := #_w31 AND NOT #SS_Input.Gripper.GripperRealState.%X30;
   #_w32 := #SS_Input.Gripper.GripperError AND #SS_Input.Gripper.GripperErrorState.%X31;
   #SS_Warning.Negative_00_31 := #_w32 AND #SS_Input.Gripper.GripperRealState.%X31;
   #SS_Warning.Positive_00_31 := #_w32 AND NOT #SS_Input.Gripper.GripperRealState.%X31;
END_REGION

REGION Network 9: Collective Error
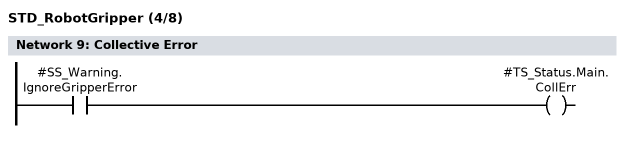
   RUNG wire#powerrail
      Contact( #SS_Warning.IgnoreGripperError )
      Coil( #TS_Status.Main.CollErr )
   END_RUNG
   // the same network as SCL:
   #TS_Status.Main.CollErr := #SS_Warning.IgnoreGripperError;
END_REGION

REGION Network 10: Collective Warning
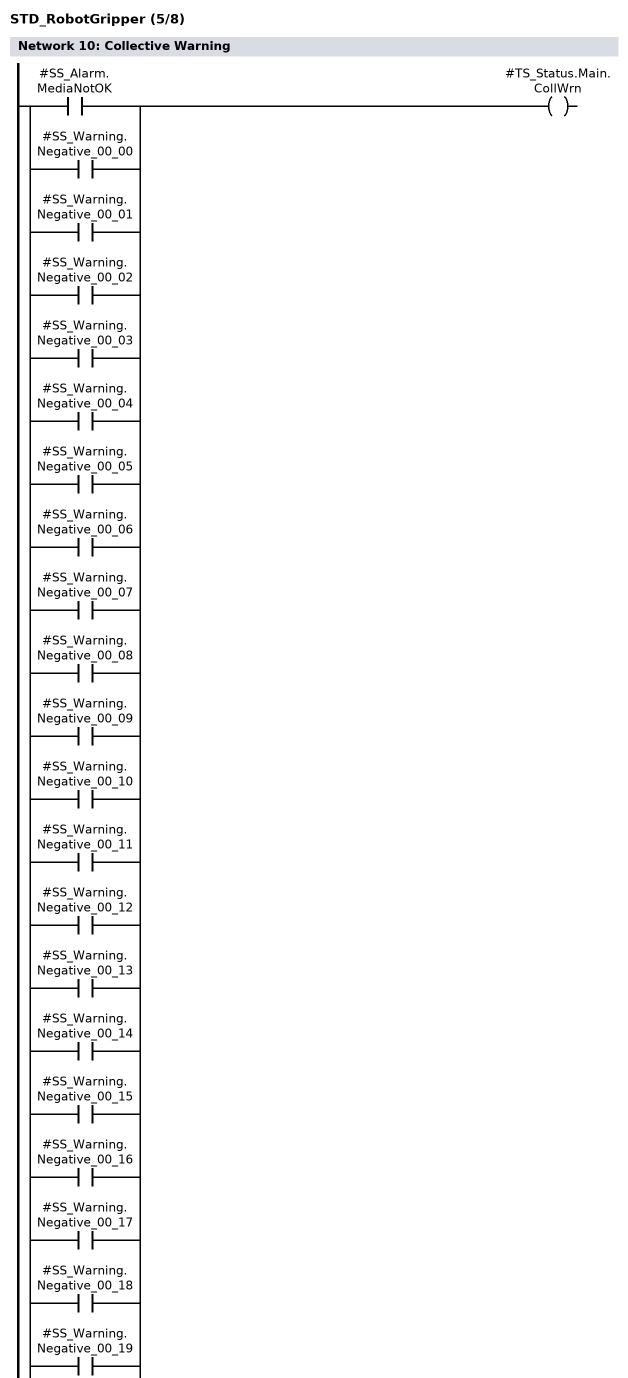
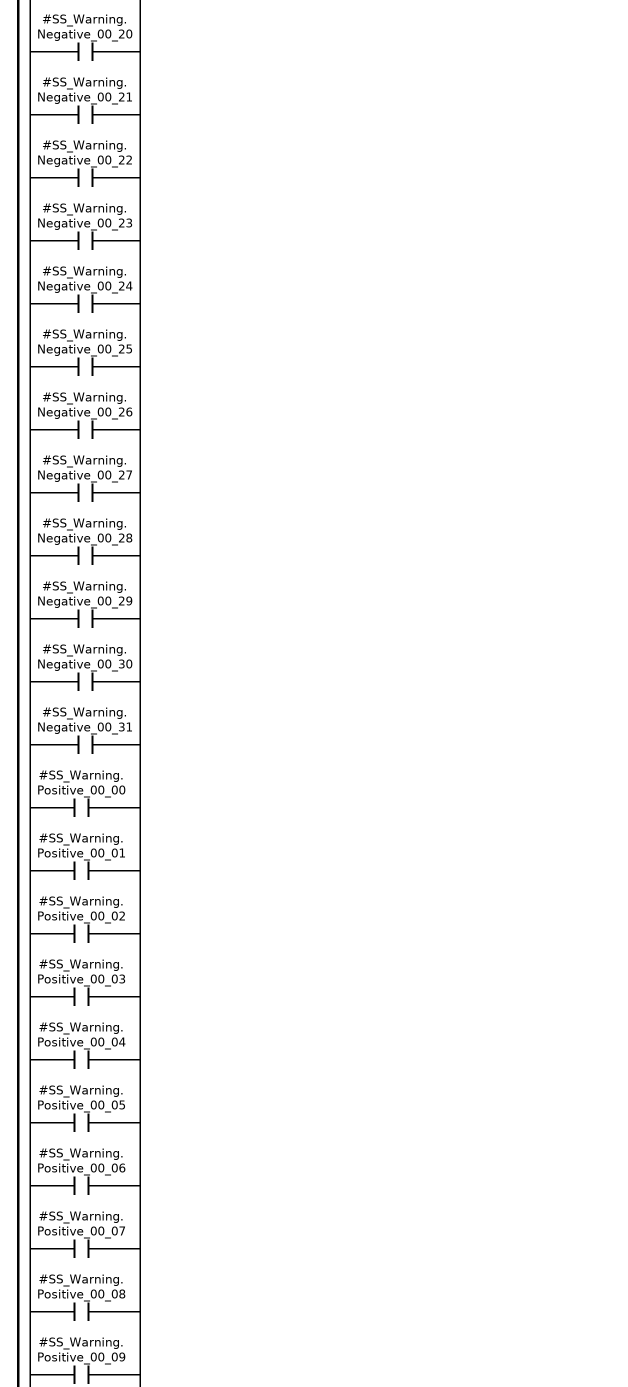
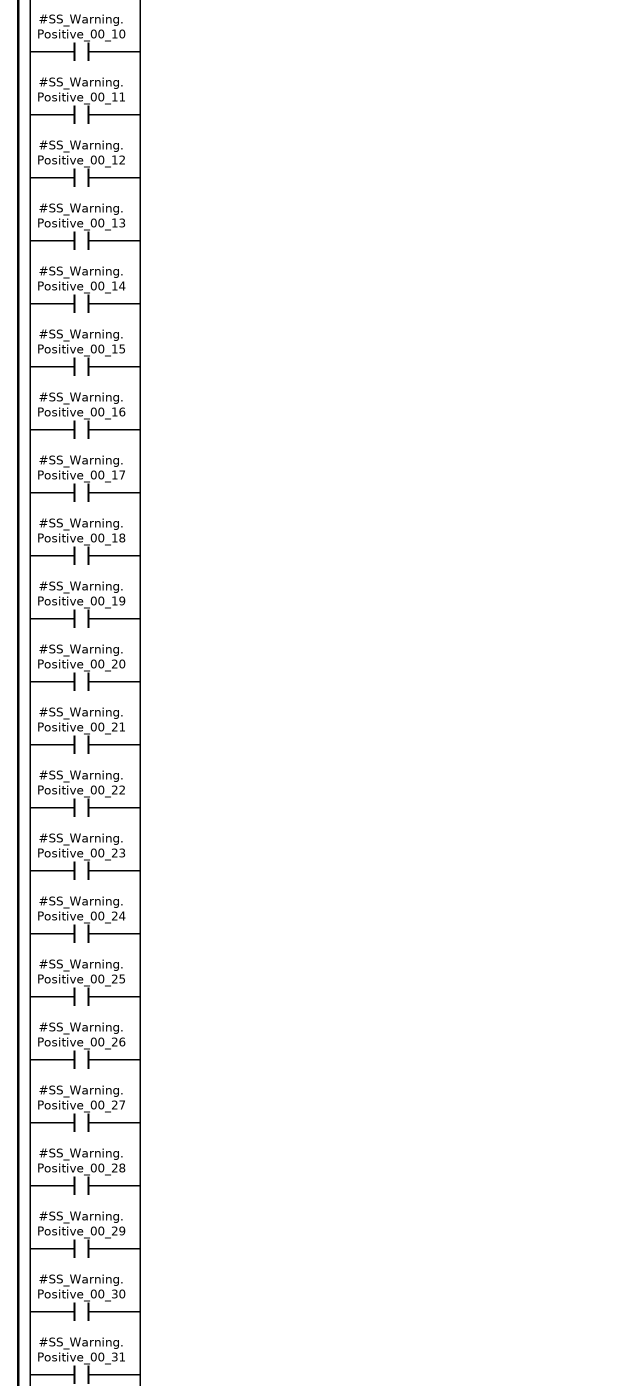
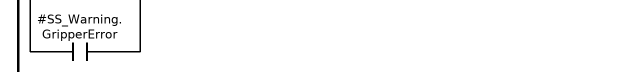
   RUNG wire#powerrail
      Contact( #SS_Alarm.MediaNotOK )
      wire#w1
      Coil( #TS_Status.Main.CollWrn )
   END_RUNG
   RUNG wire#powerrail
      Contact( #SS_Warning.Negative_00_00 )
   END_RUNG wire#w1
   RUNG wire#powerrail
      Contact( #SS_Warning.Negative_00_01 )
   END_RUNG wire#w1
   RUNG wire#powerrail
      Contact( #SS_Warning.Negative_00_02 )
   END_RUNG wire#w1
   RUNG wire#powerrail
      Contact( #SS_Warning.Negative_00_03 )
   END_RUNG wire#w1
   RUNG wire#powerrail
      Contact( #SS_Warning.Negative_00_04 )
   END_RUNG wire#w1
   RUNG wire#powerrail
      Contact( #SS_Warning.Negative_00_05 )
   END_RUNG wire#w1
   RUNG wire#powerrail
      Contact( #SS_Warning.Negative_00_06 )
   END_RUNG wire#w1
   RUNG wire#powerrail
      Contact( #SS_Warning.Negative_00_07 )
   END_RUNG wire#w1
   RUNG wire#powerrail
      Contact( #SS_Warning.Negative_00_08 )
   END_RUNG wire#w1
   RUNG wire#powerrail
      Contact( #SS_Warning.Negative_00_09 )
   END_RUNG wire#w1
   RUNG wire#powerrail
      Contact( #SS_Warning.Negative_00_10 )
   END_RUNG wire#w1
   RUNG wire#powerrail
      Contact( #SS_Warning.Negative_00_11 )
   END_RUNG wire#w1
   RUNG wire#powerrail
      Contact( #SS_Warning.Negative_00_12 )
   END_RUNG wire#w1
   RUNG wire#powerrail
      Contact( #SS_Warning.Negative_00_13 )
   END_RUNG wire#w1
   RUNG wire#powerrail
      Contact( #SS_Warning.Negative_00_14 )
   END_RUNG wire#w1
   RUNG wire#powerrail
      Contact( #SS_Warning.Negative_00_15 )
   END_RUNG wire#w1
   RUNG wire#powerrail
      Contact( #SS_Warning.Negative_00_16 )
   END_RUNG wire#w1
   RUNG wire#powerrail
      Contact( #SS_Warning.Negative_00_17 )
   END_RUNG wire#w1
   RUNG wire#powerrail
      Contact( #SS_Warning.Negative_00_18 )
   END_RUNG wire#w1
   RUNG wire#powerrail
      Contact( #SS_Warning.Negative_00_19 )
   END_RUNG wire#w1
   RUNG wire#powerrail
      Contact( #SS_Warning.Negative_00_20 )
   END_RUNG wire#w1
   RUNG wire#powerrail
      Contact( #SS_Warning.Negative_00_21 )
   END_RUNG wire#w1
   RUNG wire#powerrail
      Contact( #SS_Warning.Negative_00_22 )
   END_RUNG wire#w1
   RUNG wire#powerrail
      Contact( #SS_Warning.Negative_00_23 )
   END_RUNG wire#w1
   RUNG wire#powerrail
      Contact( #SS_Warning.Negative_00_24 )
   END_RUNG wire#w1
   RUNG wire#powerrail
      Contact( #SS_Warning.Negative_00_25 )
   END_RUNG wire#w1
   RUNG wire#powerrail
      Contact( #SS_Warning.Negative_00_26 )
   END_RUNG wire#w1
   RUNG wire#powerrail
      Contact( #SS_Warning.Negative_00_27 )
   END_RUNG wire#w1
   RUNG wire#powerrail
      Contact( #SS_Warning.Negative_00_28 )
   END_RUNG wire#w1
   RUNG wire#powerrail
      Contact( #SS_Warning.Negative_00_29 )
   END_RUNG wire#w1
   RUNG wire#powerrail
      Contact( #SS_Warning.Negative_00_30 )
   END_RUNG wire#w1
   RUNG wire#powerrail
      Contact( #SS_Warning.Negative_00_31 )
   END_RUNG wire#w1
   RUNG wire#powerrail
      Contact( #SS_Warning.Positive_00_00 )
   END_RUNG wire#w1
   RUNG wire#powerrail
      Contact( #SS_Warning.Positive_00_01 )
   END_RUNG wire#w1
   RUNG wire#powerrail
      Contact( #SS_Warning.Positive_00_02 )
   END_RUNG wire#w1
   RUNG wire#powerrail
      Contact( #SS_Warning.Positive_00_03 )
   END_RUNG wire#w1
   RUNG wire#powerrail
      Contact( #SS_Warning.Positive_00_04 )
   END_RUNG wire#w1
   RUNG wire#powerrail
      Contact( #SS_Warning.Positive_00_05 )
   END_RUNG wire#w1
   RUNG wire#powerrail
      Contact( #SS_Warning.Positive_00_06 )
   END_RUNG wire#w1
   RUNG wire#powerrail
      Contact( #SS_Warning.Positive_00_07 )
   END_RUNG wire#w1
   RUNG wire#powerrail
      Contact( #SS_Warning.Positive_00_08 )
   END_RUNG wire#w1
   RUNG wire#powerrail
      Contact( #SS_Warning.Positive_00_09 )
   END_RUNG wire#w1
   RUNG wire#powerrail
      Contact( #SS_Warning.Positive_00_10 )
   END_RUNG wire#w1
   RUNG wire#powerrail
      Contact( #SS_Warning.Positive_00_11 )
   END_RUNG wire#w1
   RUNG wire#powerrail
      Contact( #SS_Warning.Positive_00_12 )
   END_RUNG wire#w1
   RUNG wire#powerrail
      Contact( #SS_Warning.Positive_00_13 )
   END_RUNG wire#w1
   RUNG wire#powerrail
      Contact( #SS_Warning.Positive_00_14 )
   END_RUNG wire#w1
   RUNG wire#powerrail
      Contact( #SS_Warning.Positive_00_15 )
   END_RUNG wire#w1
   RUNG wire#powerrail
      Contact( #SS_Warning.Positive_00_16 )
   END_RUNG wire#w1
   RUNG wire#powerrail
      Contact( #SS_Warning.Positive_00_17 )
   END_RUNG wire#w1
   RUNG wire#powerrail
      Contact( #SS_Warning.Positive_00_18 )
   END_RUNG wire#w1
   RUNG wire#powerrail
      Contact( #SS_Warning.Positive_00_19 )
   END_RUNG wire#w1
   RUNG wire#powerrail
      Contact( #SS_Warning.Positive_00_20 )
   END_RUNG wire#w1
   RUNG wire#powerrail
      Contact( #SS_Warning.Positive_00_21 )
   END_RUNG wire#w1
   RUNG wire#powerrail
      Contact( #SS_Warning.Positive_00_22 )
   END_RUNG wire#w1
   RUNG wire#powerrail
      Contact( #SS_Warning.Positive_00_23 )
   END_RUNG wire#w1
   RUNG wire#powerrail
      Contact( #SS_Warning.Positive_00_24 )
   END_RUNG wire#w1
   RUNG wire#powerrail
      Contact( #SS_Warning.Positive_00_25 )
   END_RUNG wire#w1
   RUNG wire#powerrail
      Contact( #SS_Warning.Positive_00_26 )
   END_RUNG wire#w1
   RUNG wire#powerrail
      Contact( #SS_Warning.Positive_00_27 )
   END_RUNG wire#w1
   RUNG wire#powerrail
      Contact( #SS_Warning.Positive_00_28 )
   END_RUNG wire#w1
   RUNG wire#powerrail
      Contact( #SS_Warning.Positive_00_29 )
   END_RUNG wire#w1
   RUNG wire#powerrail
      Contact( #SS_Warning.Positive_00_30 )
   END_RUNG wire#w1
   RUNG wire#powerrail
      Contact( #SS_Warning.Positive_00_31 )
   END_RUNG wire#w1
   RUNG wire#powerrail
      Contact( #SS_Warning.GripperError )
   END_RUNG wire#w1
   // the same network as SCL:
   #TS_Status.Main.CollWrn := #SS_Alarm.MediaNotOK OR #SS_Warning.Negative_00_00 OR #SS_Warning.Negative_00_01 OR #SS_Warning.Negative_00_02 OR #SS_Warning.Negative_00_03 OR #SS_Warning.Negative_00_04 OR #SS_Warning.Negative_00_05 OR #SS_Warning.Negative_00_06 OR #SS_Warning.Negative_00_07 OR #SS_Warning.Negative_00_08 OR #SS_Warning.Negative_00_09 OR #SS_Warning.Negative_00_10 OR #SS_Warning.Negative_00_11 OR #SS_Warning.Negative_00_12 OR #SS_Warning.Negative_00_13 OR #SS_Warning.Negative_00_14 OR #SS_Warning.Negative_00_15 OR #SS_Warning.Negative_00_16 OR #SS_Warning.Negative_00_17 OR #SS_Warning.Negative_00_18 OR #SS_Warning.Negative_00_19 OR #SS_Warning.Negative_00_20 OR #SS_Warning.Negative_00_21 OR #SS_Warning.Negative_00_22 OR #SS_Warning.Negative_00_23 OR #SS_Warning.Negative_00_24 OR #SS_Warning.Negative_00_25 OR #SS_Warning.Negative_00_26 OR #SS_Warning.Negative_00_27 OR #SS_Warning.Negative_00_28 OR #SS_Warning.Negative_00_29 OR #SS_Warning.Negative_00_30 OR #SS_Warning.Negative_00_31 OR #SS_Warning.Positive_00_00 OR #SS_Warning.Positive_00_01 OR #SS_Warning.Positive_00_02 OR #SS_Warning.Positive_00_03 OR #SS_Warning.Positive_00_04 OR #SS_Warning.Positive_00_05 OR #SS_Warning.Positive_00_06 OR #SS_Warning.Positive_00_07 OR #SS_Warning.Positive_00_08 OR #SS_Warning.Positive_00_09 OR #SS_Warning.Positive_00_10 OR #SS_Warning.Positive_00_11 OR #SS_Warning.Positive_00_12 OR #SS_Warning.Positive_00_13 OR #SS_Warning.Positive_00_14 OR #SS_Warning.Positive_00_15 OR #SS_Warning.Positive_00_16 OR #SS_Warning.Positive_00_17 OR #SS_Warning.Positive_00_18 OR #SS_Warning.Positive_00_19 OR #SS_Warning.Positive_00_20 OR #SS_Warning.Positive_00_21 OR #SS_Warning.Positive_00_22 OR #SS_Warning.Positive_00_23 OR #SS_Warning.Positive_00_24 OR #SS_Warning.Positive_00_25 OR #SS_Warning.Positive_00_26 OR #SS_Warning.Positive_00_27 OR #SS_Warning.Positive_00_28 OR #SS_Warning.Positive_00_29 OR #SS_Warning.Positive_00_30 OR #SS_Warning.Positive_00_31 OR #SS_Warning.GripperError;
END_REGION

REGION Network 11: Warnings - copy to output structure
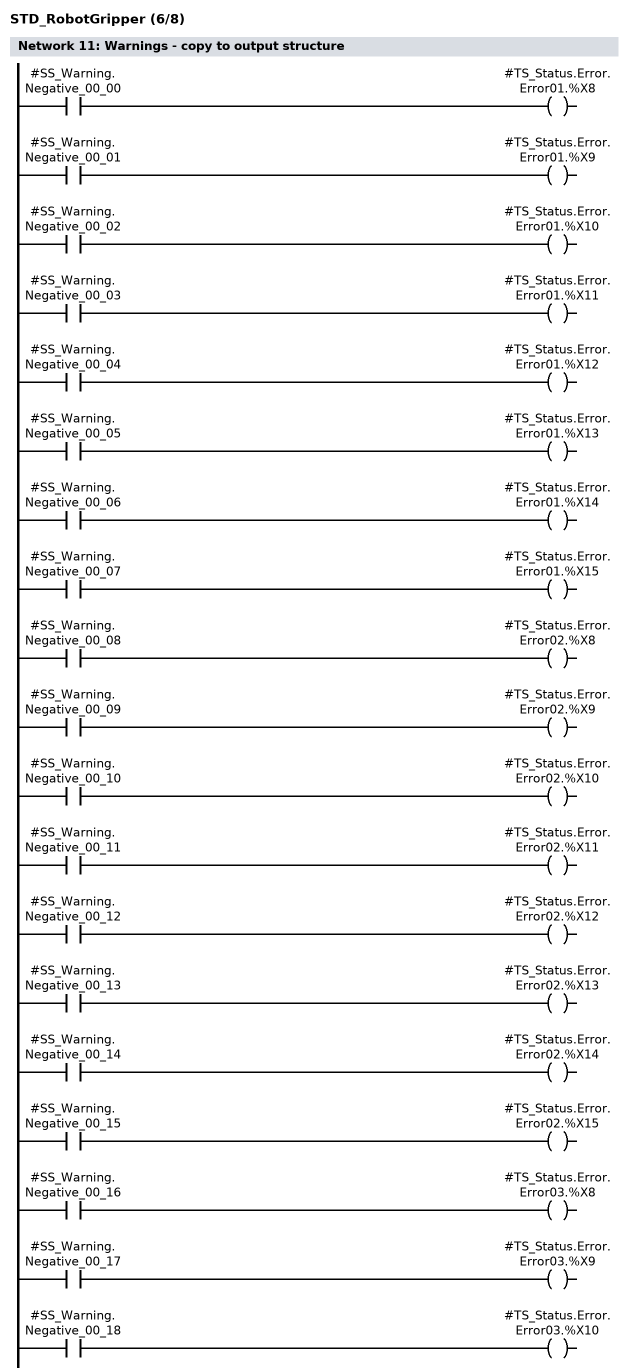
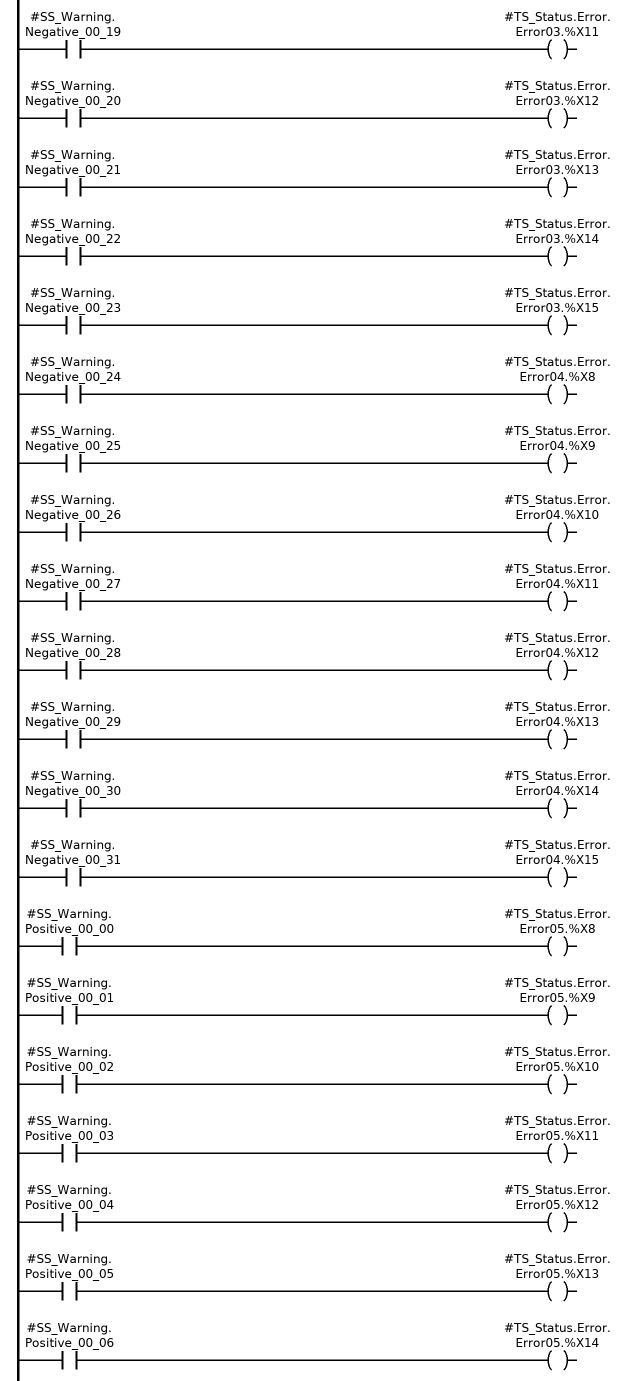
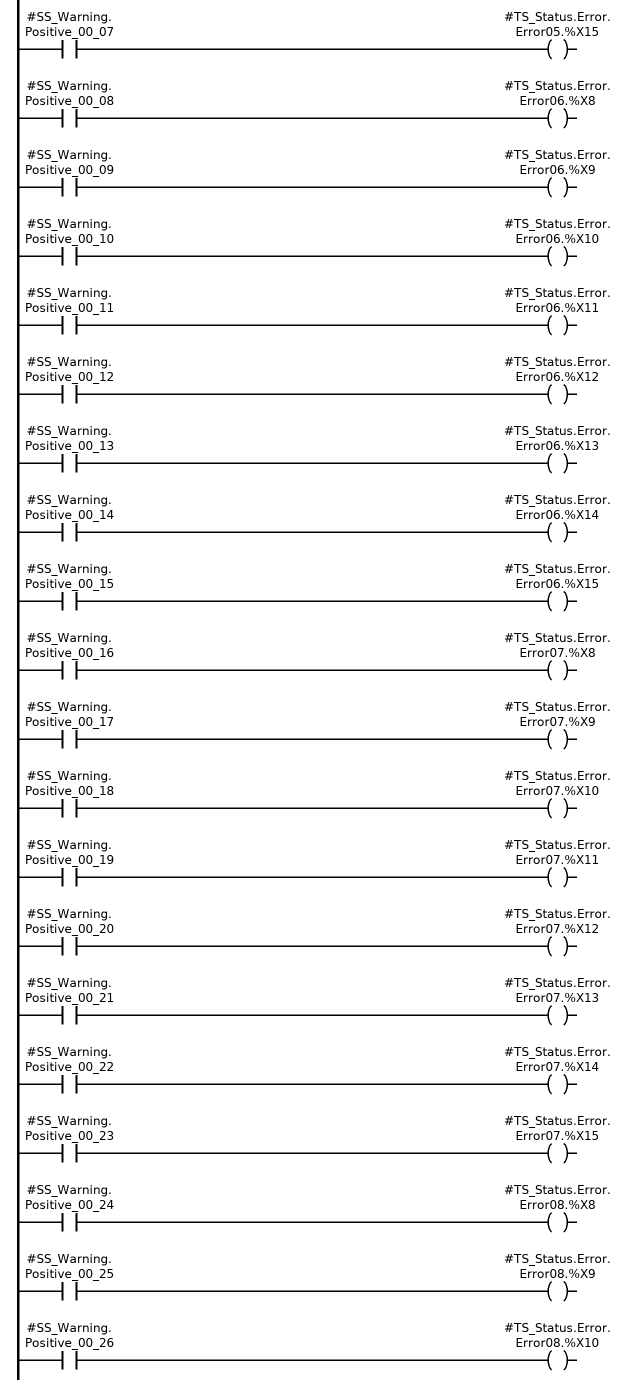
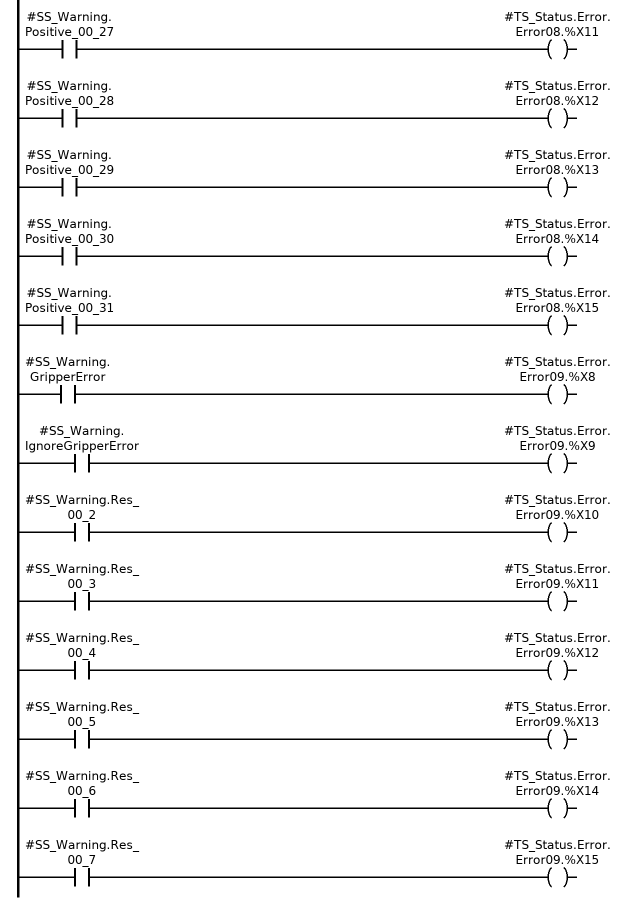
   RUNG wire#powerrail
      Contact( #SS_Warning.Negative_00_00 )
      Coil( #TS_Status.Error.Error01.%X8 )
   END_RUNG
   RUNG wire#powerrail
      Contact( #SS_Warning.Negative_00_01 )
      Coil( #TS_Status.Error.Error01.%X9 )
   END_RUNG
   RUNG wire#powerrail
      Contact( #SS_Warning.Negative_00_02 )
      Coil( #TS_Status.Error.Error01.%X10 )
   END_RUNG
   RUNG wire#powerrail
      Contact( #SS_Warning.Negative_00_03 )
      Coil( #TS_Status.Error.Error01.%X11 )
   END_RUNG
   RUNG wire#powerrail
      Contact( #SS_Warning.Negative_00_04 )
      Coil( #TS_Status.Error.Error01.%X12 )
   END_RUNG
   RUNG wire#powerrail
      Contact( #SS_Warning.Negative_00_05 )
      Coil( #TS_Status.Error.Error01.%X13 )
   END_RUNG
   RUNG wire#powerrail
      Contact( #SS_Warning.Negative_00_06 )
      Coil( #TS_Status.Error.Error01.%X14 )
   END_RUNG
   RUNG wire#powerrail
      Contact( #SS_Warning.Negative_00_07 )
      Coil( #TS_Status.Error.Error01.%X15 )
   END_RUNG
   RUNG wire#powerrail
      Contact( #SS_Warning.Negative_00_08 )
      Coil( #TS_Status.Error.Error02.%X8 )
   END_RUNG
   RUNG wire#powerrail
      Contact( #SS_Warning.Negative_00_09 )
      Coil( #TS_Status.Error.Error02.%X9 )
   END_RUNG
   RUNG wire#powerrail
      Contact( #SS_Warning.Negative_00_10 )
      Coil( #TS_Status.Error.Error02.%X10 )
   END_RUNG
   RUNG wire#powerrail
      Contact( #SS_Warning.Negative_00_11 )
      Coil( #TS_Status.Error.Error02.%X11 )
   END_RUNG
   RUNG wire#powerrail
      Contact( #SS_Warning.Negative_00_12 )
      Coil( #TS_Status.Error.Error02.%X12 )
   END_RUNG
   RUNG wire#powerrail
      Contact( #SS_Warning.Negative_00_13 )
      Coil( #TS_Status.Error.Error02.%X13 )
   END_RUNG
   RUNG wire#powerrail
      Contact( #SS_Warning.Negative_00_14 )
      Coil( #TS_Status.Error.Error02.%X14 )
   END_RUNG
   RUNG wire#powerrail
      Contact( #SS_Warning.Negative_00_15 )
      Coil( #TS_Status.Error.Error02.%X15 )
   END_RUNG
   RUNG wire#powerrail
      Contact( #SS_Warning.Negative_00_16 )
      Coil( #TS_Status.Error.Error03.%X8 )
   END_RUNG
   RUNG wire#powerrail
      Contact( #SS_Warning.Negative_00_17 )
      Coil( #TS_Status.Error.Error03.%X9 )
   END_RUNG
   RUNG wire#powerrail
      Contact( #SS_Warning.Negative_00_18 )
      Coil( #TS_Status.Error.Error03.%X10 )
   END_RUNG
   RUNG wire#powerrail
      Contact( #SS_Warning.Negative_00_19 )
      Coil( #TS_Status.Error.Error03.%X11 )
   END_RUNG
   RUNG wire#powerrail
      Contact( #SS_Warning.Negative_00_20 )
      Coil( #TS_Status.Error.Error03.%X12 )
   END_RUNG
   RUNG wire#powerrail
      Contact( #SS_Warning.Negative_00_21 )
      Coil( #TS_Status.Error.Error03.%X13 )
   END_RUNG
   RUNG wire#powerrail
      Contact( #SS_Warning.Negative_00_22 )
      Coil( #TS_Status.Error.Error03.%X14 )
   END_RUNG
   RUNG wire#powerrail
      Contact( #SS_Warning.Negative_00_23 )
      Coil( #TS_Status.Error.Error03.%X15 )
   END_RUNG
   RUNG wire#powerrail
      Contact( #SS_Warning.Negative_00_24 )
      Coil( #TS_Status.Error.Error04.%X8 )
   END_RUNG
   RUNG wire#powerrail
      Contact( #SS_Warning.Negative_00_25 )
      Coil( #TS_Status.Error.Error04.%X9 )
   END_RUNG
   RUNG wire#powerrail
      Contact( #SS_Warning.Negative_00_26 )
      Coil( #TS_Status.Error.Error04.%X10 )
   END_RUNG
   RUNG wire#powerrail
      Contact( #SS_Warning.Negative_00_27 )
      Coil( #TS_Status.Error.Error04.%X11 )
   END_RUNG
   RUNG wire#powerrail
      Contact( #SS_Warning.Negative_00_28 )
      Coil( #TS_Status.Error.Error04.%X12 )
   END_RUNG
   RUNG wire#powerrail
      Contact( #SS_Warning.Negative_00_29 )
      Coil( #TS_Status.Error.Error04.%X13 )
   END_RUNG
   RUNG wire#powerrail
      Contact( #SS_Warning.Negative_00_30 )
      Coil( #TS_Status.Error.Error04.%X14 )
   END_RUNG
   RUNG wire#powerrail
      Contact( #SS_Warning.Negative_00_31 )
      Coil( #TS_Status.Error.Error04.%X15 )
   END_RUNG
   RUNG wire#powerrail
      Contact( #SS_Warning.Positive_00_00 )
      Coil( #TS_Status.Error.Error05.%X8 )
   END_RUNG
   RUNG wire#powerrail
      Contact( #SS_Warning.Positive_00_01 )
      Coil( #TS_Status.Error.Error05.%X9 )
   END_RUNG
   RUNG wire#powerrail
      Contact( #SS_Warning.Positive_00_02 )
      Coil( #TS_Status.Error.Error05.%X10 )
   END_RUNG
   RUNG wire#powerrail
      Contact( #SS_Warning.Positive_00_03 )
      Coil( #TS_Status.Error.Error05.%X11 )
   END_RUNG
   RUNG wire#powerrail
      Contact( #SS_Warning.Positive_00_04 )
      Coil( #TS_Status.Error.Error05.%X12 )
   END_RUNG
   RUNG wire#powerrail
      Contact( #SS_Warning.Positive_00_05 )
      Coil( #TS_Status.Error.Error05.%X13 )
   END_RUNG
   RUNG wire#powerrail
      Contact( #SS_Warning.Positive_00_06 )
      Coil( #TS_Status.Error.Error05.%X14 )
   END_RUNG
   RUNG wire#powerrail
      Contact( #SS_Warning.Positive_00_07 )
      Coil( #TS_Status.Error.Error05.%X15 )
   END_RUNG
   RUNG wire#powerrail
      Contact( #SS_Warning.Positive_00_08 )
      Coil( #TS_Status.Error.Error06.%X8 )
   END_RUNG
   RUNG wire#powerrail
      Contact( #SS_Warning.Positive_00_09 )
      Coil( #TS_Status.Error.Error06.%X9 )
   END_RUNG
   RUNG wire#powerrail
      Contact( #SS_Warning.Positive_00_10 )
      Coil( #TS_Status.Error.Error06.%X10 )
   END_RUNG
   RUNG wire#powerrail
      Contact( #SS_Warning.Positive_00_11 )
      Coil( #TS_Status.Error.Error06.%X11 )
   END_RUNG
   RUNG wire#powerrail
      Contact( #SS_Warning.Positive_00_12 )
      Coil( #TS_Status.Error.Error06.%X12 )
   END_RUNG
   RUNG wire#powerrail
      Contact( #SS_Warning.Positive_00_13 )
      Coil( #TS_Status.Error.Error06.%X13 )
   END_RUNG
   RUNG wire#powerrail
      Contact( #SS_Warning.Positive_00_14 )
      Coil( #TS_Status.Error.Error06.%X14 )
   END_RUNG
   RUNG wire#powerrail
      Contact( #SS_Warning.Positive_00_15 )
      Coil( #TS_Status.Error.Error06.%X15 )
   END_RUNG
   RUNG wire#powerrail
      Contact( #SS_Warning.Positive_00_16 )
      Coil( #TS_Status.Error.Error07.%X8 )
   END_RUNG
   RUNG wire#powerrail
      Contact( #SS_Warning.Positive_00_17 )
      Coil( #TS_Status.Error.Error07.%X9 )
   END_RUNG
   RUNG wire#powerrail
      Contact( #SS_Warning.Positive_00_18 )
      Coil( #TS_Status.Error.Error07.%X10 )
   END_RUNG
   RUNG wire#powerrail
      Contact( #SS_Warning.Positive_00_19 )
      Coil( #TS_Status.Error.Error07.%X11 )
   END_RUNG
   RUNG wire#powerrail
      Contact( #SS_Warning.Positive_00_20 )
      Coil( #TS_Status.Error.Error07.%X12 )
   END_RUNG
   RUNG wire#powerrail
      Contact( #SS_Warning.Positive_00_21 )
      Coil( #TS_Status.Error.Error07.%X13 )
   END_RUNG
   RUNG wire#powerrail
      Contact( #SS_Warning.Positive_00_22 )
      Coil( #TS_Status.Error.Error07.%X14 )
   END_RUNG
   RUNG wire#powerrail
      Contact( #SS_Warning.Positive_00_23 )
      Coil( #TS_Status.Error.Error07.%X15 )
   END_RUNG
   RUNG wire#powerrail
      Contact( #SS_Warning.Positive_00_24 )
      Coil( #TS_Status.Error.Error08.%X8 )
   END_RUNG
   RUNG wire#powerrail
      Contact( #SS_Warning.Positive_00_25 )
      Coil( #TS_Status.Error.Error08.%X9 )
   END_RUNG
   RUNG wire#powerrail
      Contact( #SS_Warning.Positive_00_26 )
      Coil( #TS_Status.Error.Error08.%X10 )
   END_RUNG
   RUNG wire#powerrail
      Contact( #SS_Warning.Positive_00_27 )
      Coil( #TS_Status.Error.Error08.%X11 )
   END_RUNG
   RUNG wire#powerrail
      Contact( #SS_Warning.Positive_00_28 )
      Coil( #TS_Status.Error.Error08.%X12 )
   END_RUNG
   RUNG wire#powerrail
      Contact( #SS_Warning.Positive_00_29 )
      Coil( #TS_Status.Error.Error08.%X13 )
   END_RUNG
   RUNG wire#powerrail
      Contact( #SS_Warning.Positive_00_30 )
      Coil( #TS_Status.Error.Error08.%X14 )
   END_RUNG
   RUNG wire#powerrail
      Contact( #SS_Warning.Positive_00_31 )
      Coil( #TS_Status.Error.Error08.%X15 )
   END_RUNG
   RUNG wire#powerrail
      Contact( #SS_Warning.GripperError )
      Coil( #TS_Status.Error.Error09.%X8 )
   END_RUNG
   RUNG wire#powerrail
      Contact( #SS_Warning.IgnoreGripperError )
      Coil( #TS_Status.Error.Error09.%X9 )
   END_RUNG
   RUNG wire#powerrail
      Contact( #SS_Warning.Res_00_2 )
      Coil( #TS_Status.Error.Error09.%X10 )
   END_RUNG
   RUNG wire#powerrail
      Contact( #SS_Warning.Res_00_3 )
      Coil( #TS_Status.Error.Error09.%X11 )
   END_RUNG
   RUNG wire#powerrail
      Contact( #SS_Warning.Res_00_4 )
      Coil( #TS_Status.Error.Error09.%X12 )
   END_RUNG
   RUNG wire#powerrail
      Contact( #SS_Warning.Res_00_5 )
      Coil( #TS_Status.Error.Error09.%X13 )
   END_RUNG
   RUNG wire#powerrail
      Contact( #SS_Warning.Res_00_6 )
      Coil( #TS_Status.Error.Error09.%X14 )
   END_RUNG
   RUNG wire#powerrail
      Contact( #SS_Warning.Res_00_7 )
      Coil( #TS_Status.Error.Error09.%X15 )
   END_RUNG
   // the same network as SCL:
   #TS_Status.Error.Error01.%X8 := #SS_Warning.Negative_00_00;
   #TS_Status.Error.Error01.%X9 := #SS_Warning.Negative_00_01;
   #TS_Status.Error.Error01.%X10 := #SS_Warning.Negative_00_02;
   #TS_Status.Error.Error01.%X11 := #SS_Warning.Negative_00_03;
   #TS_Status.Error.Error01.%X12 := #SS_Warning.Negative_00_04;
   #TS_Status.Error.Error01.%X13 := #SS_Warning.Negative_00_05;
   #TS_Status.Error.Error01.%X14 := #SS_Warning.Negative_00_06;
   #TS_Status.Error.Error01.%X15 := #SS_Warning.Negative_00_07;
   #TS_Status.Error.Error02.%X8 := #SS_Warning.Negative_00_08;
   #TS_Status.Error.Error02.%X9 := #SS_Warning.Negative_00_09;
   #TS_Status.Error.Error02.%X10 := #SS_Warning.Negative_00_10;
   #TS_Status.Error.Error02.%X11 := #SS_Warning.Negative_00_11;
   #TS_Status.Error.Error02.%X12 := #SS_Warning.Negative_00_12;
   #TS_Status.Error.Error02.%X13 := #SS_Warning.Negative_00_13;
   #TS_Status.Error.Error02.%X14 := #SS_Warning.Negative_00_14;
   #TS_Status.Error.Error02.%X15 := #SS_Warning.Negative_00_15;
   #TS_Status.Error.Error03.%X8 := #SS_Warning.Negative_00_16;
   #TS_Status.Error.Error03.%X9 := #SS_Warning.Negative_00_17;
   #TS_Status.Error.Error03.%X10 := #SS_Warning.Negative_00_18;
   #TS_Status.Error.Error03.%X11 := #SS_Warning.Negative_00_19;
   #TS_Status.Error.Error03.%X12 := #SS_Warning.Negative_00_20;
   #TS_Status.Error.Error03.%X13 := #SS_Warning.Negative_00_21;
   #TS_Status.Error.Error03.%X14 := #SS_Warning.Negative_00_22;
   #TS_Status.Error.Error03.%X15 := #SS_Warning.Negative_00_23;
   #TS_Status.Error.Error04.%X8 := #SS_Warning.Negative_00_24;
   #TS_Status.Error.Error04.%X9 := #SS_Warning.Negative_00_25;
   #TS_Status.Error.Error04.%X10 := #SS_Warning.Negative_00_26;
   #TS_Status.Error.Error04.%X11 := #SS_Warning.Negative_00_27;
   #TS_Status.Error.Error04.%X12 := #SS_Warning.Negative_00_28;
   #TS_Status.Error.Error04.%X13 := #SS_Warning.Negative_00_29;
   #TS_Status.Error.Error04.%X14 := #SS_Warning.Negative_00_30;
   #TS_Status.Error.Error04.%X15 := #SS_Warning.Negative_00_31;
   #TS_Status.Error.Error05.%X8 := #SS_Warning.Positive_00_00;
   #TS_Status.Error.Error05.%X9 := #SS_Warning.Positive_00_01;
   #TS_Status.Error.Error05.%X10 := #SS_Warning.Positive_00_02;
   #TS_Status.Error.Error05.%X11 := #SS_Warning.Positive_00_03;
   #TS_Status.Error.Error05.%X12 := #SS_Warning.Positive_00_04;
   #TS_Status.Error.Error05.%X13 := #SS_Warning.Positive_00_05;
   #TS_Status.Error.Error05.%X14 := #SS_Warning.Positive_00_06;
   #TS_Status.Error.Error05.%X15 := #SS_Warning.Positive_00_07;
   #TS_Status.Error.Error06.%X8 := #SS_Warning.Positive_00_08;
   #TS_Status.Error.Error06.%X9 := #SS_Warning.Positive_00_09;
   #TS_Status.Error.Error06.%X10 := #SS_Warning.Positive_00_10;
   #TS_Status.Error.Error06.%X11 := #SS_Warning.Positive_00_11;
   #TS_Status.Error.Error06.%X12 := #SS_Warning.Positive_00_12;
   #TS_Status.Error.Error06.%X13 := #SS_Warning.Positive_00_13;
   #TS_Status.Error.Error06.%X14 := #SS_Warning.Positive_00_14;
   #TS_Status.Error.Error06.%X15 := #SS_Warning.Positive_00_15;
   #TS_Status.Error.Error07.%X8 := #SS_Warning.Positive_00_16;
   #TS_Status.Error.Error07.%X9 := #SS_Warning.Positive_00_17;
   #TS_Status.Error.Error07.%X10 := #SS_Warning.Positive_00_18;
   #TS_Status.Error.Error07.%X11 := #SS_Warning.Positive_00_19;
   #TS_Status.Error.Error07.%X12 := #SS_Warning.Positive_00_20;
   #TS_Status.Error.Error07.%X13 := #SS_Warning.Positive_00_21;
   #TS_Status.Error.Error07.%X14 := #SS_Warning.Positive_00_22;
   #TS_Status.Error.Error07.%X15 := #SS_Warning.Positive_00_23;
   #TS_Status.Error.Error08.%X8 := #SS_Warning.Positive_00_24;
   #TS_Status.Error.Error08.%X9 := #SS_Warning.Positive_00_25;
   #TS_Status.Error.Error08.%X10 := #SS_Warning.Positive_00_26;
   #TS_Status.Error.Error08.%X11 := #SS_Warning.Positive_00_27;
   #TS_Status.Error.Error08.%X12 := #SS_Warning.Positive_00_28;
   #TS_Status.Error.Error08.%X13 := #SS_Warning.Positive_00_29;
   #TS_Status.Error.Error08.%X14 := #SS_Warning.Positive_00_30;
   #TS_Status.Error.Error08.%X15 := #SS_Warning.Positive_00_31;
   #TS_Status.Error.Error09.%X8 := #SS_Warning.GripperError;
   #TS_Status.Error.Error09.%X9 := #SS_Warning.IgnoreGripperError;
   #TS_Status.Error.Error09.%X10 := #SS_Warning.Res_00_2;
   #TS_Status.Error.Error09.%X11 := #SS_Warning.Res_00_3;
   #TS_Status.Error.Error09.%X12 := #SS_Warning.Res_00_4;
   #TS_Status.Error.Error09.%X13 := #SS_Warning.Res_00_5;
   #TS_Status.Error.Error09.%X14 := #SS_Warning.Res_00_6;
   #TS_Status.Error.Error09.%X15 := #SS_Warning.Res_00_7;
END_REGION

REGION Network 12: Gripper State copy
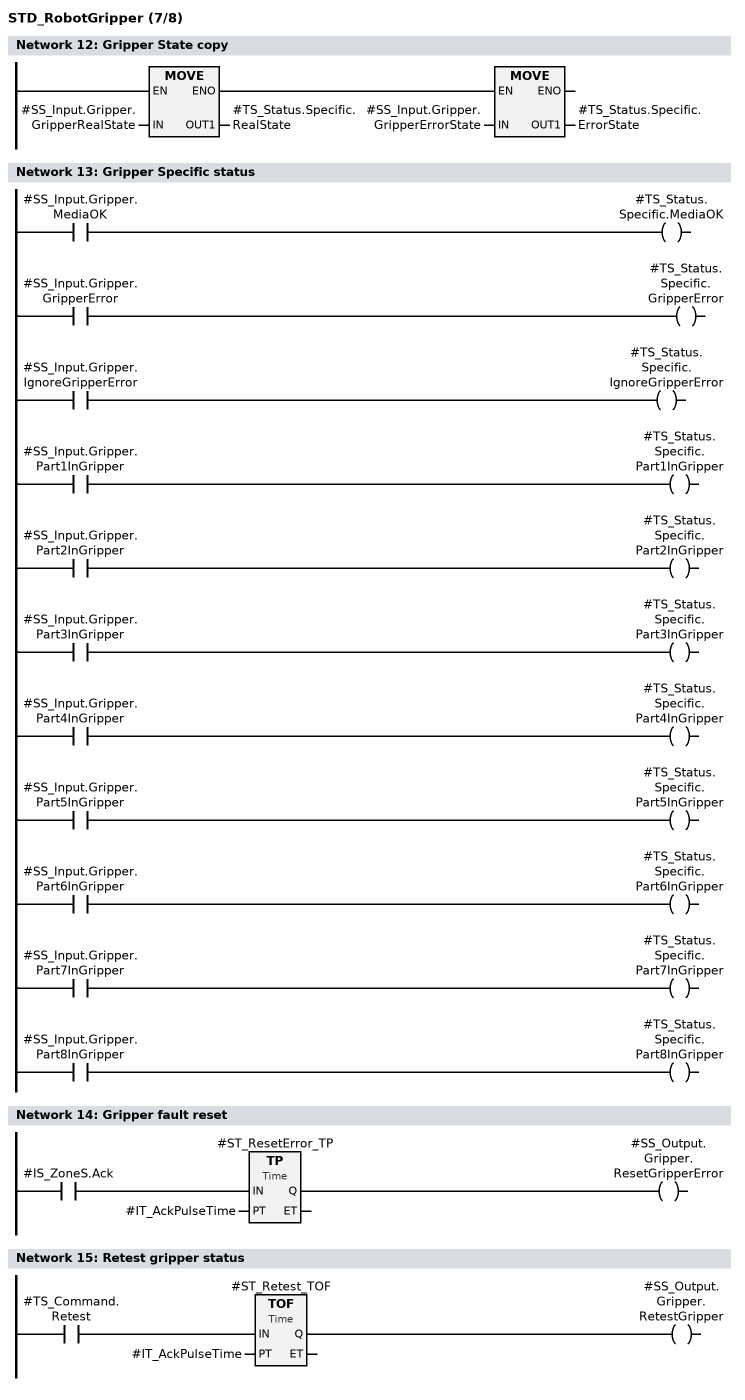
   RUNG wire#powerrail
      Move(in := #SS_Input.Gripper.GripperRealState, out1 => #TS_Status.Specific.RealState)
      Move(in := #SS_Input.Gripper.GripperErrorState, out1 => #TS_Status.Specific.ErrorState)
   END_RUNG
   // the same network as SCL:
   #TS_Status.Specific.RealState := #SS_Input.Gripper.GripperRealState;
   #TS_Status.Specific.ErrorState := #SS_Input.Gripper.GripperErrorState;
END_REGION

REGION Network 13: Gripper Specific status
   RUNG wire#powerrail
      Contact( #SS_Input.Gripper.MediaOK )
      Coil( #TS_Status.Specific.MediaOK )
   END_RUNG
   RUNG wire#powerrail
      Contact( #SS_Input.Gripper.GripperError )
      Coil( #TS_Status.Specific.GripperError )
   END_RUNG
   RUNG wire#powerrail
      Contact( #SS_Input.Gripper.IgnoreGripperError )
      Coil( #TS_Status.Specific.IgnoreGripperError )
   END_RUNG
   RUNG wire#powerrail
      Contact( #SS_Input.Gripper.Part1InGripper )
      Coil( #TS_Status.Specific.Part1InGripper )
   END_RUNG
   RUNG wire#powerrail
      Contact( #SS_Input.Gripper.Part2InGripper )
      Coil( #TS_Status.Specific.Part2InGripper )
   END_RUNG
   RUNG wire#powerrail
      Contact( #SS_Input.Gripper.Part3InGripper )
      Coil( #TS_Status.Specific.Part3InGripper )
   END_RUNG
   RUNG wire#powerrail
      Contact( #SS_Input.Gripper.Part4InGripper )
      Coil( #TS_Status.Specific.Part4InGripper )
   END_RUNG
   RUNG wire#powerrail
      Contact( #SS_Input.Gripper.Part5InGripper )
      Coil( #TS_Status.Specific.Part5InGripper )
   END_RUNG
   RUNG wire#powerrail
      Contact( #SS_Input.Gripper.Part6InGripper )
      Coil( #TS_Status.Specific.Part6InGripper )
   END_RUNG
   RUNG wire#powerrail
      Contact( #SS_Input.Gripper.Part7InGripper )
      Coil( #TS_Status.Specific.Part7InGripper )
   END_RUNG
   RUNG wire#powerrail
      Contact( #SS_Input.Gripper.Part8InGripper )
      Coil( #TS_Status.Specific.Part8InGripper )
   END_RUNG
   // the same network as SCL:
   #TS_Status.Specific.MediaOK := #SS_Input.Gripper.MediaOK;
   #TS_Status.Specific.GripperError := #SS_Input.Gripper.GripperError;
   #TS_Status.Specific.IgnoreGripperError := #SS_Input.Gripper.IgnoreGripperError;
   #TS_Status.Specific.Part1InGripper := #SS_Input.Gripper.Part1InGripper;
   #TS_Status.Specific.Part2InGripper := #SS_Input.Gripper.Part2InGripper;
   #TS_Status.Specific.Part3InGripper := #SS_Input.Gripper.Part3InGripper;
   #TS_Status.Specific.Part4InGripper := #SS_Input.Gripper.Part4InGripper;
   #TS_Status.Specific.Part5InGripper := #SS_Input.Gripper.Part5InGripper;
   #TS_Status.Specific.Part6InGripper := #SS_Input.Gripper.Part6InGripper;
   #TS_Status.Specific.Part7InGripper := #SS_Input.Gripper.Part7InGripper;
   #TS_Status.Specific.Part8InGripper := #SS_Input.Gripper.Part8InGripper;
END_REGION

REGION Network 14: Gripper fault reset
   RUNG wire#powerrail
      Contact( #IS_ZoneS.Ack )
      { S7_Templates := "time_type := Time" } #ST_ResetError_TP.TP(pt := #IT_AckPulseTime, et =>)
      Coil( #SS_Output.Gripper.ResetGripperError )
   END_RUNG
   // the same network as SCL:
   #ST_ResetError_TP(IN := #IS_ZoneS.Ack, PT := #IT_AckPulseTime);   // TP
   #SS_Output.Gripper.ResetGripperError := #ST_ResetError_TP.Q;
END_REGION

REGION Network 15: Retest gripper status
   RUNG wire#powerrail
      Contact( #TS_Command.Retest )
      { S7_Templates := "time_type := Time" } #ST_Retest_TOF.TOF(pt := #IT_AckPulseTime, et =>)
      Coil( #SS_Output.Gripper.RetestGripper )
   END_RUNG
   // the same network as SCL:
   #ST_Retest_TOF(IN := #TS_Command.Retest, PT := #IT_AckPulseTime);   // TOF
   #SS_Output.Gripper.RetestGripper := #ST_Retest_TOF.Q;
END_REGION

REGION Network 16: Retry gripper action
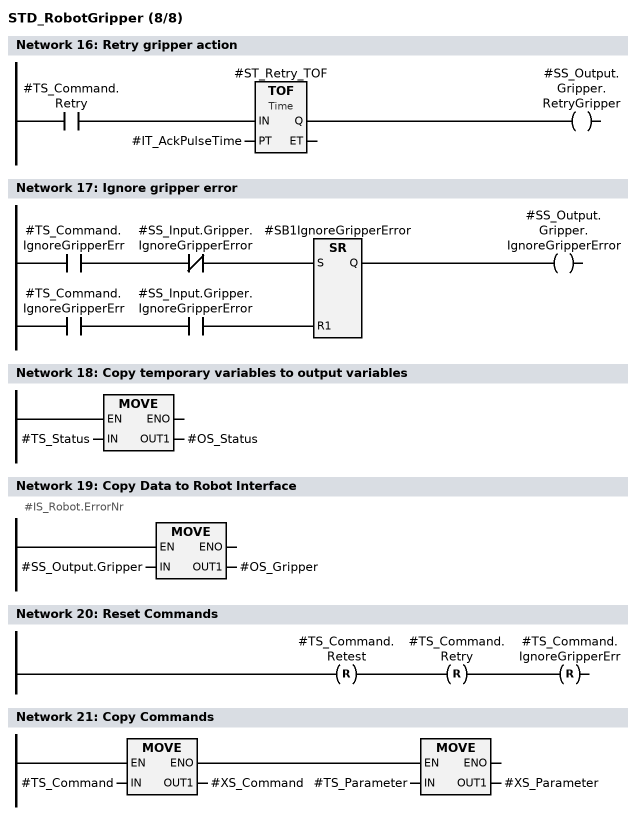
   RUNG wire#powerrail
      Contact( #TS_Command.Retry )
      { S7_Templates := "time_type := Time" } #ST_Retry_TOF.TOF(pt := #IT_AckPulseTime, et =>)
      Coil( #SS_Output.Gripper.RetryGripper )
   END_RUNG
   // the same network as SCL:
   #ST_Retry_TOF(IN := #TS_Command.Retry, PT := #IT_AckPulseTime);   // TOF
   #SS_Output.Gripper.RetryGripper := #ST_Retry_TOF.Q;
END_REGION

REGION Network 17: Ignore gripper error
   RUNG wire#powerrail
      Contact( #TS_Command.IgnoreGripperErr )
      I_Contact( #SS_Input.Gripper.IgnoreGripperError )
      S_SR(operand := #SB1IgnoreGripperError, r1 := wire#w1)
      Coil( #SS_Output.Gripper.IgnoreGripperError )
   END_RUNG
   RUNG wire#powerrail
      Contact( #TS_Command.IgnoreGripperErr )
      Contact( #SS_Input.Gripper.IgnoreGripperError )
   END_RUNG wire#w1
   // the same network as SCL:
   IF #TS_Command.IgnoreGripperErr AND NOT #SS_Input.Gripper.IgnoreGripperError THEN
       #SB1IgnoreGripperError := TRUE;   // SR flip-flop
   END_IF;
   IF #TS_Command.IgnoreGripperErr AND #SS_Input.Gripper.IgnoreGripperError THEN
       #SB1IgnoreGripperError := FALSE;
   END_IF;
   #SS_Output.Gripper.IgnoreGripperError := #SB1IgnoreGripperError;
END_REGION

REGION Network 18: Copy temporary variables to output variables
   RUNG wire#powerrail
      Move(in := #TS_Status, out1 => #OS_Status)
   END_RUNG
   // the same network as SCL:
   #OS_Status := #TS_Status;
END_REGION

REGION Network 19: Copy Data to Robot Interface
   // #IS_Robot.ErrorNr
   RUNG wire#powerrail
      Move(in := #SS_Output.Gripper, out1 => #OS_Gripper)
   END_RUNG
   // the same network as SCL:
   #OS_Gripper := #SS_Output.Gripper;
END_REGION

REGION Network 20: Reset Commands
   RUNG wire#powerrail
      R_Coil( #TS_Command.Retest )
      R_Coil( #TS_Command.Retry )
      R_Coil( #TS_Command.IgnoreGripperErr )
   END_RUNG
   // the same network as SCL:
   #TS_Command.Retest := FALSE;
   #TS_Command.Retry := FALSE;
   #TS_Command.IgnoreGripperErr := FALSE;
END_REGION

REGION Network 21: Copy Commands
   RUNG wire#powerrail
      Move(in := #TS_Command, out1 => #XS_Command)
      Move(in := #TS_Parameter, out1 => #XS_Parameter)
   END_RUNG
   // the same network as SCL:
   #XS_Command := #TS_Command;
   #XS_Parameter := #TS_Parameter;
END_REGION

NETWORK
TITLE = Save RLO in BR bit. The BR bit helps to implement the EN/ENO mechanism for block calls.
      SET;
      SAVE;
      BE;
END_FUNCTION_BLOCK
